QRS_NEXT_CUT()
PTP {E1 29336.998,E2 29336.998}
PTP {X 0,Y 607.858,A -85,B 0,C 180,E1 29336.998,E2 29336.998,E3 0,E4 0,E5 0,E6 0}
QRS_SPEED_INIT()
LIN {X 0,Y 607.858,Z 779,A -85,B 0,C 180,E1 29336.998,E2 29336.998,E3 0,E4 0,E5 0,E6 0} C_VEL
LIN {X 0,Y 607.858,Z 285.152,A -85,B 0,C 180,E1 29336.998,E2 29336.998} C_VEL
LIN {X 0,Y 607.858,Z 277.075,A -85,B 0,C 180,E1 29336.998,E2 29336.998} C_VEL
LIN {X 0,Y 607.845,Z 275.075,A -85,B 0,C 180,E1 29336.81,E2 29336.81} C_VEL
LIN {X 0,Y 607.872,Z 275.077,A -85,B 0,C 180,E1 29333.959,E2 29333.959} C_VEL
LIN {X 0,Y 607.849,Z 275.075,A -85,B 0,C 180,E1 29330.82,E2 29330.82} C_VEL
LIN {X 0,Y 607.873,Z 275.077,A -85,B 0,C 180,E1 29327.944,E2 29327.944} C_VEL
LIN {X 0,Y 607.848,Z 275.075,A -85,B 0,C 180,E1 29324.743,E2 29324.743} C_VEL
LIN {X 0,Y 607.877,Z 275.077,A -85,B 0,C 180,E1 29321.89,E2 29321.89} C_VEL
LIN {X 0,Y 607.853,Z 275.075,A -85,B 0,C 180,E1 29318.786,E2 29318.786} C_VEL
LIN {X 0,Y 607.875,Z 275.077,A -85,B 0,C 180,E1 29315.905,E2 29315.905} C_VEL
LIN {X 0,Y 607.85,Z 275.075,A -85,B 0,C 180,E1 29312.684,E2 29312.684} C_VEL
LIN {X 0,Y 607.895,Z 275.077,A -85,B 0,C 180,E1 29309.711,E2 29309.711} C_VEL
LIN {X 0,Y 607.853,Z 275.074,A -85,B 0,C 180,E1 29306.677,E2 29306.677} C_VEL
LIN {X 0,Y 607.897,Z 275.077,A -85,B 0,C 180,E1 29303.695,E2 29303.695} C_VEL
LIN {X 0,Y 607.852,Z 275.074,A -85,B 0,C 180,E1 29300.588,E2 29300.588} C_VEL
LIN {X 0,Y 607.905,Z 275.078,A -85,B 0,C 180,E1 29297.599,E2 29297.599} C_VEL
LIN {X 0,Y 607.851,Z 275.074,A -85,B 0,C 180,E1 29294.484,E2 29294.484} C_VEL
LIN {X 0,Y 607.918,Z 275.075,A -85,B 0,C 180,E1 29291.389,E2 29291.389} C_VEL
LIN {X 0,Y 607.852,Z 275.075,A -85,B 0,C 180,E1 29288.318,E2 29288.318} C_VEL
LIN {X 0,Y 607.91,Z 275.072,A -85,B 0,C 180,E1 29285.175,E2 29285.175} C_VEL
LIN {X 0,Y 607.858,Z 275.075,A -85,B 0,C 180,E1 29282.105,E2 29282.105} C_VEL
LIN {X 0,Y 607.887,Z 275.072,A -85,B 0,C 180,E1 29278.918,E2 29278.918} C_VEL
LIN {X 0,Y 607.867,Z 275.076,A -85,B 0,C 180,E1 29275.946,E2 29275.946} C_VEL
LIN {X 0,Y 607.866,Z 275.073,A -85,B 0,C 180,E1 29272.637,E2 29272.637} C_VEL
LIN {X 0,Y 607.899,Z 275.077,A -85,B 0,C 180,E1 29269.604,E2 29269.604} C_VEL
LIN {X 0,Y 607.859,Z 275.073,A -85,B 0,C 180,E1 29266.434,E2 29266.434} C_VEL
LIN {X 0,Y 607.914,Z 275.077,A -85,B 0,C 180,E1 29263.409,E2 29263.409} C_VEL
LIN {X 0,Y 607.859,Z 275.073,A -85,B 0,C 180,E1 29260.328,E2 29260.328} C_VEL
LIN {X 0,Y 607.917,Z 275.074,A -85,B 0,C 180,E1 29257.275,E2 29257.275} C_VEL
LIN {X 0,Y 607.859,Z 275.074,A -85,B 0,C 180,E1 29254.15,E2 29254.15} C_VEL
LIN {X 0,Y 607.912,Z 275.071,A -85,B 0,C 180,E1 29251.036,E2 29251.036} C_VEL
LIN {X 0,Y 607.868,Z 275.075,A -85,B 0,C 180,E1 29247.925,E2 29247.925} C_VEL
LIN {X 0,Y 607.888,Z 275.071,A -85,B 0,C 180,E1 29244.714,E2 29244.714} C_VEL
LIN {X 0,Y 607.885,Z 275.076,A -85,B 0,C 180,E1 29241.677,E2 29241.677} C_VEL
LIN {X 0,Y 607.869,Z 275.072,A -85,B 0,C 180,E1 29238.423,E2 29238.423} C_VEL
LIN {X 0,Y 607.918,Z 275.077,A -85,B 0,C 180,E1 29235.327,E2 29235.327} C_VEL
LIN {X 0,Y 607.865,Z 275.073,A -85,B 0,C 180,E1 29232.184,E2 29232.184} C_VEL
LIN {X 0,Y 607.915,Z 275.073,A -85,B 0,C 180,E1 29229.089,E2 29229.089} C_VEL
LIN {X 0,Y 607.866,Z 275.074,A -85,B 0,C 180,E1 29226.028,E2 29226.028} C_VEL
LIN {X 0,Y 607.913,Z 275.07,A -85,B 0,C 180,E1 29222.896,E2 29222.896} C_VEL
LIN {X 0,Y 607.876,Z 275.075,A -85,B 0,C 180,E1 29219.779,E2 29219.779} C_VEL
LIN {X 0,Y 607.884,Z 275.071,A -85,B 0,C 180,E1 29216.499,E2 29216.499} C_VEL
LIN {X 0,Y 607.915,Z 275.077,A -85,B 0,C 180,E1 29213.341,E2 29213.341} C_VEL
LIN {X 0,Y 607.871,Z 275.072,A -85,B 0,C 180,E1 29210.184,E2 29210.184} C_VEL
LIN {X 0,Y 607.913,Z 275.073,A -85,B 0,C 180,E1 29207.043,E2 29207.043} C_VEL
LIN {X 0,Y 607.872,Z 275.073,A -85,B 0,C 180,E1 29203.908,E2 29203.908} C_VEL
LIN {X 0,Y 607.915,Z 275.068,A -85,B 0,C 180,E1 29200.692,E2 29200.692} C_VEL
LIN {X 0,Y 607.896,Z 275.076,A -85,B 0,C 180,E1 29197.484,E2 29197.484} C_VEL
LIN {X 0,Y 607.878,Z 275.071,A -85,B 0,C 180,E1 29194.229,E2 29194.229} C_VEL
LIN {X 0,Y 607.914,Z 275.075,A -85,B 0,C 180,E1 29191.092,E2 29191.092} C_VEL
LIN {X 0,Y 607.874,Z 275.073,A -85,B 0,C 180,E1 29187.953,E2 29187.953} C_VEL
LIN {X 0,Y 607.888,Z 275.253,A -85,B 0,C 180,E1 29186.335,E2 29186.335} C_VEL
LIN {X 0,Y 607.91,Z 304.241,A -85,B 0,C 180,E1 29183.248,E2 29183.248} C_VEL
LIN {X 0,Y 607.905,Z 334.622,A -85,B 0,C 180,E1 29180.088,E2 29180.088} C_VEL
LIN {X 0,Y 607.882,Z 364.695,A -85,B 0,C 180,E1 29177.023,E2 29177.023} C_VEL
LIN {X 0,Y 607.92,Z 399.027,A -85,B 0,C 180,E1 29173.581,E2 29173.581} C_VEL
LIN {X 0,Y 607.897,Z 405.045,A -85,B 0,C 180,E1 29173.009,E2 29173.009} C_VEL
LIN {X 0,Y 607.911,Z 516.068,A -85,B 0,C 180,E1 29171.67,E2 29171.67} C_VEL
LIN {X 0,Y 607.905,Z 531.255,A -85,B 0,C 180,E1 29171.31,E2 29171.31} C_VEL
LIN {X 0,Y 607.911,Z 546.081,A -85,B 0,C 180,E1 29170.757,E2 29170.757} C_VEL
LIN {X 0,Y 607.897,Z 559.139,A -85,B 0,C 180,E1 29170.087,E2 29170.087} C_VEL
LIN {X 0,Y 607.919,Z 571.341,A -85,B 0,C 180,E1 29169.274,E2 29169.274} C_VEL
LIN {X 0,Y 607.919,Z 583.519,A -85,B 0,C 180,E1 29168.225,E2 29168.225} C_VEL
LIN {X 0,Y 607.919,Z 593.771,A -85,B 0,C 180,E1 29167.084,E2 29167.084} C_VEL
LIN {X 0,Y 607.917,Z 601.752,A -85,B 0,C 180,E1 29165.946,E2 29165.946} C_VEL
LIN {X 0,Y 607.914,Z 608.844,A -85,B 0,C 180,E1 29164.621,E2 29164.621} C_VEL
LIN {X 0,Y 607.917,Z 614.161,A -85,B 0,C 180,E1 29163.204,E2 29163.204} C_VEL
LIN {X 0,Y 607.915,Z 617.299,A -85,B 0,C 180,E1 29161.884,E2 29161.884} C_VEL
LIN {X 0,Y 607.918,Z 618.88,A -85,B 0,C 180,E1 29160.47,E2 29160.47} C_VEL
LIN {X 0,Y 607.915,Z 618.551,A -85,B 0,C 180,E1 29158.962,E2 29158.962} C_VEL
LIN {X 0,Y 607.916,Z 616.35,A -85,B 0,C 180,E1 29157.548,E2 29157.548} C_VEL
LIN {X 0,Y 607.918,Z 612.603,A -85,B 0,C 180,E1 29156.227,E2 29156.227} C_VEL
LIN {X 0,Y 607.917,Z 606.529,A -85,B 0,C 180,E1 29154.809,E2 29154.809} C_VEL
LIN {X 0,Y 607.918,Z 599.252,A -85,B 0,C 180,E1 29153.577,E2 29153.577} C_VEL
LIN {X 0,Y 607.918,Z 590.573,A -85,B 0,C 180,E1 29152.438,E2 29152.438} C_VEL
LIN {X 0,Y 607.919,Z 579.903,A -85,B 0,C 180,E1 29151.344,E2 29151.344} C_VEL
LIN {X 0,Y 607.911,Z 567.267,A -85,B 0,C 180,E1 29150.341,E2 29150.341} C_VEL
LIN {X 0,Y 607.909,Z 554.716,A -85,B 0,C 180,E1 29149.575,E2 29149.575} C_VEL
LIN {X 0,Y 607.907,Z 541.317,A -85,B 0,C 180,E1 29148.952,E2 29148.952} C_VEL
LIN {X 0,Y 607.913,Z 526.652,A -85,B 0,C 180,E1 29148.472,E2 29148.472} C_VEL
LIN {X 0,Y 607.902,Z 511.857,A -85,B 0,C 180,E1 29148.173,E2 29148.173} C_VEL
LIN {X 0,Y 607.896,Z 404.579,A -85,B 0,C 180,E1 29146.88,E2 29146.88} C_VEL
LIN {X 0,Y 607.909,Z 372.874,A -85,B 0,C 180,E1 29143.713,E2 29143.713} C_VEL
LIN {X 0,Y 607.9,Z 341.655,A -85,B 0,C 180,E1 29140.544,E2 29140.544} C_VEL
LIN {X 0,Y 607.843,Z 311.899,A -85,B 0,C 180,E1 29137.463,E2 29137.463} C_VEL
LIN {X 0,Y 607.918,Z 283.604,A -85,B 0,C 180,E1 29134.473,E2 29134.473} C_VEL
LIN {X 0,Y 607.859,Z 275.078,A -85,B 0,C 180,E1 29133.527,E2 29133.527} C_VEL
LIN {X 0,Y 607.916,Z 275.071,A -85,B 0,C 180,E1 29130.434,E2 29130.434} C_VEL
LIN {X 0,Y 607.895,Z 275.076,A -85,B 0,C 180,E1 29127.238,E2 29127.238} C_VEL
LIN {X 0,Y 607.897,Z 275.07,A -85,B 0,C 180,E1 29124.022,E2 29124.022} C_VEL
LIN {X 0,Y 607.901,Z 275.074,A -85,B 0,C 180,E1 29120.927,E2 29120.927} C_VEL
LIN {X 0,Y 607.902,Z 275.072,A -85,B 0,C 180,E1 29117.85,E2 29117.85} C_VEL
LIN {X 0,Y 607.886,Z 275.072,A -85,B 0,C 180,E1 29114.748,E2 29114.748} C_VEL
LIN {X 0,Y 607.905,Z 275.077,A -85,B 0,C 180,E1 29111.517,E2 29111.517} C_VEL
LIN {X 0,Y 607.903,Z 275.071,A -85,B 0,C 180,E1 29108.32,E2 29108.32} C_VEL
LIN {X 0,Y 607.854,Z 275.076,A -85,B 0,C 180,E1 29105.15,E2 29105.15} C_VEL
LIN {X 0,Y 607.918,Z 275.077,A -85,B 0,C 180,E1 29102.09,E2 29102.09} C_VEL
LIN {X 0,Y 607.866,Z 275.304,A -85,B 0,C 180,E1 29099.751,E2 29099.751} C_VEL
LIN {X 0,Y 607.899,Z 318.111,A -85,B 0,C 180,E1 29096.84,E2 29096.84} C_VEL
LIN {X 0,Y 607.901,Z 364.581,A -85,B 0,C 180,E1 29093.765,E2 29093.765} C_VEL
LIN {X 0,Y 607.908,Z 387.125,A -85,B 0,C 180,E1 29092.324,E2 29092.324} C_VEL
LIN {X 0,Y 607.914,Z 596.287,A -85,B 0,C 180,E1 29089.705,E2 29089.705} C_VEL
LIN {X 0,Y 607.913,Z 614.57,A -85,B 0,C 180,E1 29089.305,E2 29089.305} C_VEL
LIN {X 0,Y 607.915,Z 633.394,A -85,B 0,C 180,E1 29088.707,E2 29088.707} C_VEL
LIN {X 0,Y 607.916,Z 651.048,A -85,B 0,C 180,E1 29087.963,E2 29087.963} C_VEL
LIN {X 0,Y 607.919,Z 667.781,A -85,B 0,C 180,E1 29087.073,E2 29087.073} C_VEL
LIN {X 0,Y 607.916,Z 683.634,A -85,B 0,C 180,E1 29086.041,E2 29086.041} C_VEL
LIN {X 0,Y 607.917,Z 698.556,A -85,B 0,C 180,E1 29084.868,E2 29084.868} C_VEL
LIN {X 0,Y 607.918,Z 712.22,A -85,B 0,C 180,E1 29083.582,E2 29083.582} C_VEL
LIN {X 0,Y 607.916,Z 724.902,A -85,B 0,C 180,E1 29082.154,E2 29082.154} C_VEL
LIN {X 0,Y 607.911,Z 736.22,A -85,B 0,C 180,E1 29080.616,E2 29080.616} C_VEL
LIN {X 0,Y 607.92,Z 745.986,A -85,B 0,C 180,E1 29078.99,E2 29078.99} C_VEL
LIN {X 0,Y 607.913,Z 753.852,A -85,B 0,C 180,E1 29077.352,E2 29077.352} C_VEL
LIN {X 0,Y 607.906,Z 760.105,A -85,B 0,C 180,E1 29075.664,E2 29075.664} C_VEL
LIN {X 0,Y 607.917,Z 764.871,A -85,B 0,C 180,E1 29073.867,E2 29073.867} C_VEL
LIN {X 0,Y 607.911,Z 767.786,A -85,B 0,C 180,E1 29072.074,E2 29072.074} C_VEL
LIN {X 0,Y 607.907,Z 768.939,A -85,B 0,C 180,E1 29070.283,E2 29070.283} C_VEL
LIN {X 0,Y 607.916,Z 768.348,A -85,B 0,C 180,E1 29068.493,E2 29068.493} C_VEL
LIN {X 0,Y 607.908,Z 766.006,A -85,B 0,C 180,E1 29066.701,E2 29066.701} C_VEL
LIN {X 0,Y 607.918,Z 762.098,A -85,B 0,C 180,E1 29065,E2 29065} C_VEL
LIN {X 0,Y 607.91,Z 756.47,A -85,B 0,C 180,E1 29063.295,E2 29063.295} C_VEL
LIN {X 0,Y 607.914,Z 749.426,A -85,B 0,C 180,E1 29061.679,E2 29061.679} C_VEL
LIN {X 0,Y 607.914,Z 740.513,A -85,B 0,C 180,E1 29060.056,E2 29060.056} C_VEL
LIN {X 0,Y 607.919,Z 730.15,A -85,B 0,C 180,E1 29058.522,E2 29058.522} C_VEL
LIN {X 0,Y 607.915,Z 718.352,A -85,B 0,C 180,E1 29057.075,E2 29057.075} C_VEL
LIN {X 0,Y 607.915,Z 705.096,A -85,B 0,C 180,E1 29055.718,E2 29055.718} C_VEL
LIN {X 0,Y 607.917,Z 690.243,A -85,B 0,C 180,E1 29054.45,E2 29054.45} C_VEL
LIN {X 0,Y 607.917,Z 674.23,A -85,B 0,C 180,E1 29053.322,E2 29053.322} C_VEL
LIN {X 0,Y 607.911,Z 658.041,A -85,B 0,C 180,E1 29052.385,E2 29052.385} C_VEL
LIN {X 0,Y 607.913,Z 641.082,A -85,B 0,C 180,E1 29051.592,E2 29051.592} C_VEL
LIN {X 0,Y 607.916,Z 623.251,A -85,B 0,C 180,E1 29050.946,E2 29050.946} C_VEL
LIN {X 0,Y 607.91,Z 604.277,A -85,B 0,C 180,E1 29050.449,E2 29050.449} C_VEL
LIN {X 0,Y 607.914,Z 584.868,A -85,B 0,C 180,E1 29050.129,E2 29050.129} C_VEL
LIN {X 0,Y 607.907,Z 386.276,A -85,B 0,C 180,E1 29047.646,E2 29047.646} C_VEL
LIN {X 0,Y 607.897,Z 339.401,A -85,B 0,C 180,E1 29044.579,E2 29044.579} C_VEL
LIN {X 0,Y 607.883,Z 294.506,A -85,B 0,C 180,E1 29041.565,E2 29041.565} C_VEL
LIN {X 0,Y 607.864,Z 275.08,A -85,B 0,C 180,E1 29040.216,E2 29040.216} C_VEL
LIN {X 0,Y 607.84,Z 275.078,A -85,B 0,C 180,E1 29037.125,E2 29037.125} C_VEL
LIN {X 0,Y 607.847,Z 275.077,A -85,B 0,C 180,E1 29034.35,E2 29034.35} C_VEL
LIN {X 0,Y 607.837,Z 275.077,A -85,B 0,C 180,E1 29031.084,E2 29031.084} C_VEL
LIN {X 0,Y 607.854,Z 275.077,A -85,B 0,C 180,E1 29028.228,E2 29028.228} C_VEL
LIN {X 0,Y 607.833,Z 275.077,A -85,B 0,C 180,E1 29025.019,E2 29025.019} C_VEL
LIN {X 0,Y 607.849,Z 275.077,A -85,B 0,C 180,E1 29022.252,E2 29022.252} C_VEL
LIN {X 0,Y 607.838,Z 275.077,A -85,B 0,C 180,E1 29019.052,E2 29019.052} C_VEL
LIN {X 0,Y 607.843,Z 275.077,A -85,B 0,C 180,E1 29016.293,E2 29016.293} C_VEL
LIN {X 0,Y 607.845,Z 275.077,A -85,B 0,C 180,E1 29013.102,E2 29013.102} C_VEL
LIN {X 0,Y 607.842,Z 275.077,A -85,B 0,C 180,E1 29010.332,E2 29010.332} C_VEL
LIN {X 0,Y 607.84,Z 275.077,A -85,B 0,C 180,E1 29007.002,E2 29007.002} C_VEL
LIN {X 0,Y 607.846,Z 275.077,A -85,B 0,C 180,E1 29004.283,E2 29004.283} C_VEL
LIN {X 0,Y 607.845,Z 275.076,A -85,B 0,C 180,E1 29001.015,E2 29001.015} C_VEL
LIN {X 0,Y 607.851,Z 275.077,A -85,B 0,C 180,E1 28998.213,E2 28998.213} C_VEL
LIN {X 0,Y 607.845,Z 275.076,A -85,B 0,C 180,E1 28994.967,E2 28994.967} C_VEL
LIN {X 0,Y 607.847,Z 275.077,A -85,B 0,C 180,E1 28992.252,E2 28992.252} C_VEL
LIN {X 0,Y 607.85,Z 275.076,A -85,B 0,C 180,E1 28988.991,E2 28988.991} C_VEL
LIN {X 0,Y 607.849,Z 275.077,A -85,B 0,C 180,E1 28986.234,E2 28986.234} C_VEL
LIN {X 0,Y 607.849,Z 275.076,A -85,B 0,C 180,E1 28982.924,E2 28982.924} C_VEL
LIN {X 0,Y 607.859,Z 275.077,A -85,B 0,C 180,E1 28980.096,E2 28980.096} C_VEL
LIN {X 0,Y 607.85,Z 275.075,A -85,B 0,C 180,E1 28976.89,E2 28976.89} C_VEL
LIN {X 0,Y 607.845,Z 275.075,A -85,B 0,C 180,E1 28976.81,E2 28976.81} C_VEL
LIN {X 0,Y 606.844,Z 275.204,A -85,B 0,C 180,E1 28976.084,E2 28976.084} C_VEL
LIN {X 0,Y 600.488,Z 276.008,A -85,B 0,C 180,E1 28974.046,E2 28974.046} C_VEL
LIN {X 0,Y 599.975,Z 276.065,A -85,B 0,C 180,E1 28973.517,E2 28973.517} C_VEL
LIN {X 0,Y 599.903,Z 276.065,A -85,B 0,C 180,E1 28970.504,E2 28970.504} C_VEL
LIN {X 0,Y 599.969,Z 276.063,A -85,B 0,C 180,E1 28967.392,E2 28967.392} C_VEL
LIN {X 0,Y 599.907,Z 276.065,A -85,B 0,C 180,E1 28964.337,E2 28964.337} C_VEL
LIN {X 0,Y 599.95,Z 276.063,A -85,B 0,C 180,E1 28961.19,E2 28961.19} C_VEL
LIN {X 0,Y 599.909,Z 276.065,A -85,B 0,C 180,E1 28958.286,E2 28958.286} C_VEL
LIN {X 0,Y 599.952,Z 276.062,A -85,B 0,C 180,E1 28955.169,E2 28955.169} C_VEL
LIN {X 0,Y 599.914,Z 276.065,A -85,B 0,C 180,E1 28952.184,E2 28952.184} C_VEL
LIN {X 0,Y 599.928,Z 276.063,A -85,B 0,C 180,E1 28948.894,E2 28948.894} C_VEL
LIN {X 0,Y 599.932,Z 276.065,A -85,B 0,C 180,E1 28945.924,E2 28945.924} C_VEL
LIN {X 0,Y 599.921,Z 276.063,A -85,B 0,C 180,E1 28942.774,E2 28942.774} C_VEL
LIN {X 0,Y 599.94,Z 276.065,A -85,B 0,C 180,E1 28939.839,E2 28939.839} C_VEL
LIN {X 0,Y 599.915,Z 276.063,A -85,B 0,C 180,E1 28936.606,E2 28936.606} C_VEL
LIN {X 0,Y 599.972,Z 276.067,A -85,B 0,C 180,E1 28933.54,E2 28933.54} C_VEL
LIN {X 0,Y 599.913,Z 276.063,A -85,B 0,C 180,E1 28930.392,E2 28930.392} C_VEL
LIN {X 0,Y 599.977,Z 276.063,A -85,B 0,C 180,E1 28927.343,E2 28927.343} C_VEL
LIN {X 0,Y 599.915,Z 276.064,A -85,B 0,C 180,E1 28924.247,E2 28924.247} C_VEL
LIN {X 0,Y 599.968,Z 276.061,A -85,B 0,C 180,E1 28921.105,E2 28921.105} C_VEL
LIN {X 0,Y 599.923,Z 276.064,A -85,B 0,C 180,E1 28918.033,E2 28918.033} C_VEL
LIN {X 0,Y 599.933,Z 276.061,A -85,B 0,C 180,E1 28914.728,E2 28914.728} C_VEL
LIN {X 0,Y 599.948,Z 276.065,A -85,B 0,C 180,E1 28911.713,E2 28911.713} C_VEL
LIN {X 0,Y 599.923,Z 276.062,A -85,B 0,C 180,E1 28908.509,E2 28908.509} C_VEL
LIN {X 0,Y 599.975,Z 276.066,A -85,B 0,C 180,E1 28905.464,E2 28905.464} C_VEL
LIN {X 0,Y 599.92,Z 276.063,A -85,B 0,C 180,E1 28902.317,E2 28902.317} C_VEL
LIN {X 0,Y 599.978,Z 276.062,A -85,B 0,C 180,E1 28899.205,E2 28899.205} C_VEL
LIN {X 0,Y 599.922,Z 276.063,A -85,B 0,C 180,E1 28896.122,E2 28896.122} C_VEL
LIN {X 0,Y 599.971,Z 276.059,A -85,B 0,C 180,E1 28892.961,E2 28892.961} C_VEL
LIN {X 0,Y 599.93,Z 276.064,A -85,B 0,C 180,E1 28889.904,E2 28889.904} C_VEL
LIN {X 0,Y 599.939,Z 276.06,A -85,B 0,C 180,E1 28886.607,E2 28886.607} C_VEL
LIN {X 0,Y 599.965,Z 276.066,A -85,B 0,C 180,E1 28883.492,E2 28883.492} C_VEL
LIN {X 0,Y 599.926,Z 276.062,A -85,B 0,C 180,E1 28880.309,E2 28880.309} C_VEL
LIN {X 0,Y 599.977,Z 276.063,A -85,B 0,C 180,E1 28877.194,E2 28877.194} C_VEL
LIN {X 0,Y 599.926,Z 276.063,A -85,B 0,C 180,E1 28874.071,E2 28874.071} C_VEL
LIN {X 0,Y 599.974,Z 276.059,A -85,B 0,C 180,E1 28870.885,E2 28870.885} C_VEL
LIN {X 0,Y 599.938,Z 276.064,A -85,B 0,C 180,E1 28867.77,E2 28867.77} C_VEL
LIN {X 0,Y 599.937,Z 276.06,A -85,B 0,C 180,E1 28864.427,E2 28864.427} C_VEL
LIN {X 0,Y 599.974,Z 276.067,A -85,B 0,C 180,E1 28861.317,E2 28861.317} C_VEL
LIN {X 0,Y 599.929,Z 276.062,A -85,B 0,C 180,E1 28858.107,E2 28858.107} C_VEL
LIN {X 0,Y 599.975,Z 276.061,A -85,B 0,C 180,E1 28855.02,E2 28855.02} C_VEL
LIN {X 0,Y 599.933,Z 276.063,A -85,B 0,C 180,E1 28851.869,E2 28851.869} C_VEL
LIN {X 0,Y 599.968,Z 276.058,A -85,B 0,C 180,E1 28848.704,E2 28848.704} C_VEL
LIN {X 0,Y 599.957,Z 276.065,A -85,B 0,C 180,E1 28845.499,E2 28845.499} C_VEL
LIN {X 0,Y 599.938,Z 276.06,A -85,B 0,C 180,E1 28842.27,E2 28842.27} C_VEL
LIN {X 0,Y 599.977,Z 276.065,A -85,B 0,C 180,E1 28839.166,E2 28839.166} C_VEL
LIN {X 0,Y 599.934,Z 276.062,A -85,B 0,C 180,E1 28836.035,E2 28836.035} C_VEL
LIN {X 0,Y 599.974,Z 276.06,A -85,B 0,C 180,E1 28832.868,E2 28832.868} C_VEL
LIN {X 0,Y 599.94,Z 276.064,A -85,B 0,C 180,E1 28829.738,E2 28829.738} C_VEL
LIN {X 0,Y 599.997,Z 276.241,A -85,B 0,C 180,E1 28826.601,E2 28826.601} C_VEL
LIN {X 0,Y 600.264,Z 284.48,A -85,B 0,C 180,E1 28825.69,E2 28825.69} C_VEL
LIN {X 0,Y 600.192,Z 314.246,A -85,B 0,C 180,E1 28822.501,E2 28822.501} C_VEL
LIN {X 0,Y 600.105,Z 344.224,A -85,B 0,C 180,E1 28819.362,E2 28819.362} C_VEL
LIN {X 0,Y 600.059,Z 375.427,A -85,B 0,C 180,E1 28816.155,E2 28816.155} C_VEL
LIN {X 0,Y 600.035,Z 405.097,A -85,B 0,C 180,E1 28813.182,E2 28813.182} C_VEL
LIN {X 0,Y 600.074,Z 516.391,A -85,B 0,C 180,E1 28811.819,E2 28811.819} C_VEL
LIN {X 0,Y 600.051,Z 531.275,A -85,B 0,C 180,E1 28811.46,E2 28811.46} C_VEL
LIN {X 0,Y 600.03,Z 546.096,A -85,B 0,C 180,E1 28810.9,E2 28810.9} C_VEL
LIN {X 0,Y 599.988,Z 559.151,A -85,B 0,C 180,E1 28810.221,E2 28810.221} C_VEL
LIN {X 0,Y 599.986,Z 571.349,A -85,B 0,C 180,E1 28809.398,E2 28809.398} C_VEL
LIN {X 0,Y 599.961,Z 583.526,A -85,B 0,C 180,E1 28808.335,E2 28808.335} C_VEL
LIN {X 0,Y 599.942,Z 593.776,A -85,B 0,C 180,E1 28807.179,E2 28807.179} C_VEL
LIN {X 0,Y 599.928,Z 601.756,A -85,B 0,C 180,E1 28806.026,E2 28806.026} C_VEL
LIN {X 0,Y 599.919,Z 608.863,A -85,B 0,C 180,E1 28804.679,E2 28804.679} C_VEL
LIN {X 0,Y 599.92,Z 614.164,A -85,B 0,C 180,E1 28803.247,E2 28803.247} C_VEL
LIN {X 0,Y 599.916,Z 617.301,A -85,B 0,C 180,E1 28801.909,E2 28801.909} C_VEL
LIN {X 0,Y 599.919,Z 618.88,A -85,B 0,C 180,E1 28800.476,E2 28800.476} C_VEL
LIN {X 0,Y 599.915,Z 618.55,A -85,B 0,C 180,E1 28798.948,E2 28798.948} C_VEL
LIN {X 0,Y 599.917,Z 616.349,A -85,B 0,C 180,E1 28797.515,E2 28797.515} C_VEL
LIN {X 0,Y 599.919,Z 612.601,A -85,B 0,C 180,E1 28796.176,E2 28796.176} C_VEL
LIN {X 0,Y 599.923,Z 606.526,A -85,B 0,C 180,E1 28794.739,E2 28794.739} C_VEL
LIN {X 0,Y 599.933,Z 599.249,A -85,B 0,C 180,E1 28793.491,E2 28793.491} C_VEL
LIN {X 0,Y 599.948,Z 590.568,A -85,B 0,C 180,E1 28792.337,E2 28792.337} C_VEL
LIN {X 0,Y 599.97,Z 579.677,A -85,B 0,C 180,E1 28791.208,E2 28791.208} C_VEL
LIN {X 0,Y 599.983,Z 567.257,A -85,B 0,C 180,E1 28790.212,E2 28790.212} C_VEL
LIN {X 0,Y 600.012,Z 554.707,A -85,B 0,C 180,E1 28789.437,E2 28789.437} C_VEL
LIN {X 0,Y 600.037,Z 541.302,A -85,B 0,C 180,E1 28788.805,E2 28788.805} C_VEL
LIN {X 0,Y 600.064,Z 525.867,A -85,B 0,C 180,E1 28788.297,E2 28788.297} C_VEL
LIN {X 0,Y 600.069,Z 510.599,A -85,B 0,C 180,E1 28787.999,E2 28787.999} C_VEL
LIN {X 0,Y 600.001,Z 404.573,A -85,B 0,C 180,E1 28786.704,E2 28786.704} C_VEL
LIN {X 0,Y 600.055,Z 372.38,A -85,B 0,C 180,E1 28783.444,E2 28783.444} C_VEL
LIN {X 0,Y 600.14,Z 341.577,A -85,B 0,C 180,E1 28780.275,E2 28780.275} C_VEL
LIN {X 0,Y 600.139,Z 312.38,A -85,B 0,C 180,E1 28777.209,E2 28777.209} C_VEL
LIN {X 0,Y 600.29,Z 284.085,A -85,B 0,C 180,E1 28774.178,E2 28774.178} C_VEL
LIN {X 0,Y 600.043,Z 276.767,A -85,B 0,C 180,E1 28773.368,E2 28773.368} C_VEL
LIN {X 0,Y 599.929,Z 276.07,A -85,B 0,C 180,E1 28773.256,E2 28773.256} C_VEL
LIN {X 0,Y 599.947,Z 276.061,A -85,B 0,C 180,E1 28770.001,E2 28770.001} C_VEL
LIN {X 0,Y 599.974,Z 276.065,A -85,B 0,C 180,E1 28766.864,E2 28766.864} C_VEL
LIN {X 0,Y 599.951,Z 276.062,A -85,B 0,C 180,E1 28763.726,E2 28763.726} C_VEL
LIN {X 0,Y 599.962,Z 276.06,A -85,B 0,C 180,E1 28760.583,E2 28760.583} C_VEL
LIN {X 0,Y 599.968,Z 276.066,A -85,B 0,C 180,E1 28757.302,E2 28757.302} C_VEL
LIN {X 0,Y 599.974,Z 276.059,A -85,B 0,C 180,E1 28754.088,E2 28754.088} C_VEL
LIN {X 0,Y 599.935,Z 276.063,A -85,B 0,C 180,E1 28750.919,E2 28750.919} C_VEL
LIN {X 0,Y 599.968,Z 276.067,A -85,B 0,C 180,E1 28747.707,E2 28747.707} C_VEL
LIN {X 0,Y 599.93,Z 276.064,A -85,B 0,C 180,E1 28744.634,E2 28744.634} C_VEL
LIN {X 0,Y 599.909,Z 276.068,A -85,B 0,C 180,E1 28741.422,E2 28741.422} C_VEL
LIN {X 0,Y 599.972,Z 276.106,A -85,B 0,C 180,E1 28740.126,E2 28740.126} C_VEL
LIN {X 0,Y 600.585,Z 279.631,A -85,B 0,C 180,E1 28739.846,E2 28739.846} C_VEL
LIN {X 0,Y 600.503,Z 321.261,A -85,B 0,C 180,E1 28736.983,E2 28736.983} C_VEL
LIN {X 0,Y 600.374,Z 367.732,A -85,B 0,C 180,E1 28733.872,E2 28733.872} C_VEL
LIN {X 0,Y 600.412,Z 387.17,A -85,B 0,C 180,E1 28732.618,E2 28732.618} C_VEL
LIN {X 0,Y 600.374,Z 596.287,A -85,B 0,C 180,E1 28729.963,E2 28729.963} C_VEL
LIN {X 0,Y 600.333,Z 615.274,A -85,B 0,C 180,E1 28729.539,E2 28729.539} C_VEL
LIN {X 0,Y 600.287,Z 633.392,A -85,B 0,C 180,E1 28728.954,E2 28728.954} C_VEL
LIN {X 0,Y 600.233,Z 651.044,A -85,B 0,C 180,E1 28728.201,E2 28728.201} C_VEL
LIN {X 0,Y 600.179,Z 667.696,A -85,B 0,C 180,E1 28727.305,E2 28727.305} C_VEL
LIN {X 0,Y 600.122,Z 683.632,A -85,B 0,C 180,E1 28726.255,E2 28726.255} C_VEL
LIN {X 0,Y 600.069,Z 698.557,A -85,B 0,C 180,E1 28725.067,E2 28725.067} C_VEL
LIN {X 0,Y 600.02,Z 712.014,A -85,B 0,C 180,E1 28723.786,E2 28723.786} C_VEL
LIN {X 0,Y 599.982,Z 724.903,A -85,B 0,C 180,E1 28722.317,E2 28722.317} C_VEL
LIN {X 0,Y 599.953,Z 736.221,A -85,B 0,C 180,E1 28720.758,E2 28720.758} C_VEL
LIN {X 0,Y 599.939,Z 745.987,A -85,B 0,C 180,E1 28719.111,E2 28719.111} C_VEL
LIN {X 0,Y 599.923,Z 754.034,A -85,B 0,C 180,E1 28717.407,E2 28717.407} C_VEL
LIN {X 0,Y 599.91,Z 760.408,A -85,B 0,C 180,E1 28715.644,E2 28715.644} C_VEL
LIN {X 0,Y 599.918,Z 764.872,A -85,B 0,C 180,E1 28713.919,E2 28713.919} C_VEL
LIN {X 0,Y 599.911,Z 767.787,A -85,B 0,C 180,E1 28712.102,E2 28712.102} C_VEL
LIN {X 0,Y 599.907,Z 768.939,A -85,B 0,C 180,E1 28710.287,E2 28710.287} C_VEL
LIN {X 0,Y 599.915,Z 768.349,A -85,B 0,C 180,E1 28708.473,E2 28708.473} C_VEL
LIN {X 0,Y 599.907,Z 766.006,A -85,B 0,C 180,E1 28706.657,E2 28706.657} C_VEL
LIN {X 0,Y 599.92,Z 762.098,A -85,B 0,C 180,E1 28704.933,E2 28704.933} C_VEL
LIN {X 0,Y 599.919,Z 756.47,A -85,B 0,C 180,E1 28703.205,E2 28703.205} C_VEL
LIN {X 0,Y 599.927,Z 749.427,A -85,B 0,C 180,E1 28701.567,E2 28701.567} C_VEL
LIN {X 0,Y 599.947,Z 740.515,A -85,B 0,C 180,E1 28699.923,E2 28699.923} C_VEL
LIN {X 0,Y 599.969,Z 730.151,A -85,B 0,C 180,E1 28698.367,E2 28698.367} C_VEL
LIN {X 0,Y 600.001,Z 718.353,A -85,B 0,C 180,E1 28696.902,E2 28696.902} C_VEL
LIN {X 0,Y 600.046,Z 704.766,A -85,B 0,C 180,E1 28695.494,E2 28695.494} C_VEL
LIN {X 0,Y 600.103,Z 690.243,A -85,B 0,C 180,E1 28694.242,E2 28694.242} C_VEL
LIN {X 0,Y 600.165,Z 674.233,A -85,B 0,C 180,E1 28693.1,E2 28693.1} C_VEL
LIN {X 0,Y 600.216,Z 657.049,A -85,B 0,C 180,E1 28692.102,E2 28692.102} C_VEL
LIN {X 0,Y 600.277,Z 639.677,A -85,B 0,C 180,E1 28691.294,E2 28691.294} C_VEL
LIN {X 0,Y 600.33,Z 621.682,A -85,B 0,C 180,E1 28690.649,E2 28690.649} C_VEL
LIN {X 0,Y 600.361,Z 603.347,A -85,B 0,C 180,E1 28690.174,E2 28690.174} C_VEL
LIN {X 0,Y 600.389,Z 583.667,A -85,B 0,C 180,E1 28689.854,E2 28689.854} C_VEL
LIN {X 0,Y 600.335,Z 386.634,A -85,B 0,C 180,E1 28687.372,E2 28687.372} C_VEL
LIN {X 0,Y 600.446,Z 340.976,A -85,B 0,C 180,E1 28684.346,E2 28684.346} C_VEL
LIN {X 0,Y 600.565,Z 296.568,A -85,B 0,C 180,E1 28681.329,E2 28681.329} C_VEL
LIN {X 0,Y 600.426,Z 277.965,A -85,B 0,C 180,E1 28680.029,E2 28680.029} C_VEL
LIN {X 0,Y 599.967,Z 276.066,A -85,B 0,C 180,E1 28679.844,E2 28679.844} C_VEL
LIN {X 0,Y 599.891,Z 276.067,A -85,B 0,C 180,E1 28676.794,E2 28676.794} C_VEL
LIN {X 0,Y 599.96,Z 276.068,A -85,B 0,C 180,E1 28673.729,E2 28673.729} C_VEL
LIN {X 0,Y 599.89,Z 276.067,A -85,B 0,C 180,E1 28670.809,E2 28670.809} C_VEL
LIN {X 0,Y 599.966,Z 276.067,A -85,B 0,C 180,E1 28667.681,E2 28667.681} C_VEL
LIN {X 0,Y 599.889,Z 276.067,A -85,B 0,C 180,E1 28664.698,E2 28664.698} C_VEL
LIN {X 0,Y 599.969,Z 276.067,A -85,B 0,C 180,E1 28661.678,E2 28661.678} C_VEL
LIN {X 0,Y 599.89,Z 276.066,A -85,B 0,C 180,E1 28658.685,E2 28658.685} C_VEL
LIN {X 0,Y 599.975,Z 276.066,A -85,B 0,C 180,E1 28655.682,E2 28655.682} C_VEL
LIN {X 0,Y 599.893,Z 276.066,A -85,B 0,C 180,E1 28652.572,E2 28652.572} C_VEL
LIN {X 0,Y 599.946,Z 276.065,A -85,B 0,C 180,E1 28649.449,E2 28649.449} C_VEL
LIN {X 0,Y 599.896,Z 276.066,A -85,B 0,C 180,E1 28646.49,E2 28646.49} C_VEL
LIN {X 0,Y 599.94,Z 276.065,A -85,B 0,C 180,E1 28643.37,E2 28643.37} C_VEL
LIN {X 0,Y 599.901,Z 276.066,A -85,B 0,C 180,E1 28640.387,E2 28640.387} C_VEL
LIN {X 0,Y 599.92,Z 276.065,A -85,B 0,C 180,E1 28637.158,E2 28637.158} C_VEL
LIN {X 0,Y 599.907,Z 276.066,A -85,B 0,C 180,E1 28634.282,E2 28634.282} C_VEL
LIN {X 0,Y 599.908,Z 276.065,A -85,B 0,C 180,E1 28630.954,E2 28630.954} C_VEL
LIN {X 0,Y 599.919,Z 276.066,A -85,B 0,C 180,E1 28628.12,E2 28628.12} C_VEL
LIN {X 0,Y 599.906,Z 276.065,A -85,B 0,C 180,E1 28624.877,E2 28624.877} C_VEL
LIN {X 0,Y 599.929,Z 276.066,A -85,B 0,C 180,E1 28622.007,E2 28622.007} C_VEL
LIN {X 0,Y 599.908,Z 276.064,A -85,B 0,C 180,E1 28618.855,E2 28618.855} C_VEL
LIN {X 0,Y 599.93,Z 276.066,A -85,B 0,C 180,E1 28615.988,E2 28615.988} C_VEL
LIN {X 0,Y 599.975,Z 276.065,A -85,B 0,C 180,E1 28613.517,E2 28613.517} C_VEL
LIN {X 0,Y 598.985,Z 276.182,A -85,B 0,C 180,E1 28612.781,E2 28612.781} C_VEL
LIN {X 0,Y 592.49,Z 276.989,A -85,B 0,C 180,E1 28610.718,E2 28610.718} C_VEL
LIN {X 0,Y 591.975,Z 277.054,A -85,B 0,C 180,E1 28610.18,E2 28610.18} C_VEL
LIN {X 0,Y 591.974,Z 277.053,A -85,B 0,C 180,E1 28606.821,E2 28606.821} C_VEL
LIN {X 0,Y 591.996,Z 277.055,A -85,B 0,C 180,E1 28603.921,E2 28603.921} C_VEL
LIN {X 0,Y 591.97,Z 277.053,A -85,B 0,C 180,E1 28600.669,E2 28600.669} C_VEL
LIN {X 0,Y 592.039,Z 277.055,A -85,B 0,C 180,E1 28597.564,E2 28597.564} C_VEL
LIN {X 0,Y 591.968,Z 277.053,A -85,B 0,C 180,E1 28594.413,E2 28594.413} C_VEL
LIN {X 0,Y 592.034,Z 277.052,A -85,B 0,C 180,E1 28591.341,E2 28591.341} C_VEL
LIN {X 0,Y 591.971,Z 277.053,A -85,B 0,C 180,E1 28588.315,E2 28588.315} C_VEL
LIN {X 0,Y 592.019,Z 277.051,A -85,B 0,C 180,E1 28585.164,E2 28585.164} C_VEL
LIN {X 0,Y 591.976,Z 277.053,A -85,B 0,C 180,E1 28582.188,E2 28582.188} C_VEL
LIN {X 0,Y 591.998,Z 277.051,A -85,B 0,C 180,E1 28578.931,E2 28578.931} C_VEL
LIN {X 0,Y 591.984,Z 277.054,A -85,B 0,C 180,E1 28576.013,E2 28576.013} C_VEL
LIN {X 0,Y 591.984,Z 277.051,A -85,B 0,C 180,E1 28572.72,E2 28572.72} C_VEL
LIN {X 0,Y 592.023,Z 277.055,A -85,B 0,C 180,E1 28569.638,E2 28569.638} C_VEL
LIN {X 0,Y 591.976,Z 277.052,A -85,B 0,C 180,E1 28566.478,E2 28566.478} C_VEL
LIN {X 0,Y 592.038,Z 277.054,A -85,B 0,C 180,E1 28563.404,E2 28563.404} C_VEL
LIN {X 0,Y 591.976,Z 277.052,A -85,B 0,C 180,E1 28560.331,E2 28560.331} C_VEL
LIN {X 0,Y 592.04,Z 277.05,A -85,B 0,C 180,E1 28557.236,E2 28557.236} C_VEL
LIN {X 0,Y 591.981,Z 277.053,A -85,B 0,C 180,E1 28554.125,E2 28554.125} C_VEL
LIN {X 0,Y 592.018,Z 277.049,A -85,B 0,C 180,E1 28550.946,E2 28550.946} C_VEL
LIN {X 0,Y 591.992,Z 277.053,A -85,B 0,C 180,E1 28547.901,E2 28547.901} C_VEL
LIN {X 0,Y 591.989,Z 277.051,A -85,B 0,C 180,E1 28544.575,E2 28544.575} C_VEL
LIN {X 0,Y 592.032,Z 277.055,A -85,B 0,C 180,E1 28541.494,E2 28541.494} C_VEL
LIN {X 0,Y 591.982,Z 277.051,A -85,B 0,C 180,E1 28538.351,E2 28538.351} C_VEL
LIN {X 0,Y 592.039,Z 277.052,A -85,B 0,C 180,E1 28535.232,E2 28535.232} C_VEL
LIN {X 0,Y 591.984,Z 277.052,A -85,B 0,C 180,E1 28532.129,E2 28532.129} C_VEL
LIN {X 0,Y 592.029,Z 277.049,A -85,B 0,C 180,E1 28528.935,E2 28528.935} C_VEL
LIN {X 0,Y 591.996,Z 277.053,A -85,B 0,C 180,E1 28525.834,E2 28525.834} C_VEL
LIN {X 0,Y 591.993,Z 277.05,A -85,B 0,C 180,E1 28522.471,E2 28522.471} C_VEL
LIN {X 0,Y 592.036,Z 277.056,A -85,B 0,C 180,E1 28519.377,E2 28519.377} C_VEL
LIN {X 0,Y 591.986,Z 277.051,A -85,B 0,C 180,E1 28516.197,E2 28516.197} C_VEL
LIN {X 0,Y 592.038,Z 277.051,A -85,B 0,C 180,E1 28513.113,E2 28513.113} C_VEL
LIN {X 0,Y 591.991,Z 277.052,A -85,B 0,C 180,E1 28509.948,E2 28509.948} C_VEL
LIN {X 0,Y 592.023,Z 277.048,A -85,B 0,C 180,E1 28506.721,E2 28506.721} C_VEL
LIN {X 0,Y 592.02,Z 277.054,A -85,B 0,C 180,E1 28503.517,E2 28503.517} C_VEL
LIN {X 0,Y 591.996,Z 277.049,A -85,B 0,C 180,E1 28500.338,E2 28500.338} C_VEL
LIN {X 0,Y 592.038,Z 277.052,A -85,B 0,C 180,E1 28497.171,E2 28497.171} C_VEL
LIN {X 0,Y 591.992,Z 277.051,A -85,B 0,C 180,E1 28493.996,E2 28493.996} C_VEL
LIN {X 0,Y 592.038,Z 277.047,A -85,B 0,C 180,E1 28490.817,E2 28490.817} C_VEL
LIN {X 0,Y 592.007,Z 277.053,A -85,B 0,C 180,E1 28487.632,E2 28487.632} C_VEL
LIN {X 0,Y 592.005,Z 277.048,A -85,B 0,C 180,E1 28484.361,E2 28484.361} C_VEL
LIN {X 0,Y 592.037,Z 277.054,A -85,B 0,C 180,E1 28481.194,E2 28481.194} C_VEL
LIN {X 0,Y 591.995,Z 277.051,A -85,B 0,C 180,E1 28478.056,E2 28478.056} C_VEL
LIN {X 0,Y 592.036,Z 277.05,A -85,B 0,C 180,E1 28474.923,E2 28474.923} C_VEL
LIN {X 0,Y 591.997,Z 277.052,A -85,B 0,C 180,E1 28471.798,E2 28471.798} C_VEL
LIN {X 0,Y 592.029,Z 277.049,A -85,B 0,C 180,E1 28468.549,E2 28468.549} C_VEL
LIN {X 0,Y 592.046,Z 277.139,A -85,B 0,C 180,E1 28466.89,E2 28466.89} C_VEL
LIN {X 0,Y 592.666,Z 281.437,A -85,B 0,C 180,E1 28466.384,E2 28466.384} C_VEL
LIN {X 0,Y 592.523,Z 309.616,A -85,B 0,C 180,E1 28463.308,E2 28463.308} C_VEL
LIN {X 0,Y 592.379,Z 340.33,A -85,B 0,C 180,E1 28460.036,E2 28460.036} C_VEL
LIN {X 0,Y 592.241,Z 372.02,A -85,B 0,C 180,E1 28456.727,E2 28456.727} C_VEL
LIN {X 0,Y 592.11,Z 404.162,A -85,B 0,C 180,E1 28453.428,E2 28453.428} C_VEL
LIN {X 0,Y 592.176,Z 405.374,A -85,B 0,C 180,E1 28453.358,E2 28453.358} C_VEL
LIN {X 0,Y 592.241,Z 516.485,A -85,B 0,C 180,E1 28451.977,E2 28451.977} C_VEL
LIN {X 0,Y 592.201,Z 531.295,A -85,B 0,C 180,E1 28451.614,E2 28451.614} C_VEL
LIN {X 0,Y 592.153,Z 546.112,A -85,B 0,C 180,E1 28451.047,E2 28451.047} C_VEL
LIN {X 0,Y 592.084,Z 559.163,A -85,B 0,C 180,E1 28450.359,E2 28450.359} C_VEL
LIN {X 0,Y 592.057,Z 571.56,A -85,B 0,C 180,E1 28449.509,E2 28449.509} C_VEL
LIN {X 0,Y 592.006,Z 583.532,A -85,B 0,C 180,E1 28448.448,E2 28448.448} C_VEL
LIN {X 0,Y 591.966,Z 593.78,A -85,B 0,C 180,E1 28447.276,E2 28447.276} C_VEL
LIN {X 0,Y 591.94,Z 601.761,A -85,B 0,C 180,E1 28446.107,E2 28446.107} C_VEL
LIN {X 0,Y 591.926,Z 608.849,A -85,B 0,C 180,E1 28444.746,E2 28444.746} C_VEL
LIN {X 0,Y 591.922,Z 614.166,A -85,B 0,C 180,E1 28443.291,E2 28443.291} C_VEL
LIN {X 0,Y 591.916,Z 617.302,A -85,B 0,C 180,E1 28441.935,E2 28441.935} C_VEL
LIN {X 0,Y 591.919,Z 618.881,A -85,B 0,C 180,E1 28440.483,E2 28440.483} C_VEL
LIN {X 0,Y 591.914,Z 618.549,A -85,B 0,C 180,E1 28438.934,E2 28438.934} C_VEL
LIN {X 0,Y 591.918,Z 616.348,A -85,B 0,C 180,E1 28437.482,E2 28437.482} C_VEL
LIN {X 0,Y 591.921,Z 612.599,A -85,B 0,C 180,E1 28436.124,E2 28436.124} C_VEL
LIN {X 0,Y 591.93,Z 606.523,A -85,B 0,C 180,E1 28434.668,E2 28434.668} C_VEL
LIN {X 0,Y 591.948,Z 599.245,A -85,B 0,C 180,E1 28433.403,E2 28433.403} C_VEL
LIN {X 0,Y 591.978,Z 590.562,A -85,B 0,C 180,E1 28432.233,E2 28432.233} C_VEL
LIN {X 0,Y 592.021,Z 579.978,A -85,B 0,C 180,E1 28431.118,E2 28431.118} C_VEL
LIN {X 0,Y 592.059,Z 567.611,A -85,B 0,C 180,E1 28430.107,E2 28430.107} C_VEL
LIN {X 0,Y 592.118,Z 554.698,A -85,B 0,C 180,E1 28429.294,E2 28429.294} C_VEL
LIN {X 0,Y 592.169,Z 541.288,A -85,B 0,C 180,E1 28428.654,E2 28428.654} C_VEL
LIN {X 0,Y 592.222,Z 525.844,A -85,B 0,C 180,E1 28428.14,E2 28428.14} C_VEL
LIN {X 0,Y 592.241,Z 510.445,A -85,B 0,C 180,E1 28427.837,E2 28427.837} C_VEL
LIN {X 0,Y 592.11,Z 404.676,A -85,B 0,C 180,E1 28426.534,E2 28426.534} C_VEL
LIN {X 0,Y 592.212,Z 372.16,A -85,B 0,C 180,E1 28423.196,E2 28423.196} C_VEL
LIN {X 0,Y 592.373,Z 341.643,A -85,B 0,C 180,E1 28420.013,E2 28420.013} C_VEL
LIN {X 0,Y 592.446,Z 312.861,A -85,B 0,C 180,E1 28416.949,E2 28416.949} C_VEL
LIN {X 0,Y 592.666,Z 283.64,A -85,B 0,C 180,E1 28413.767,E2 28413.767} C_VEL
LIN {X 0,Y 592.44,Z 278.875,A -85,B 0,C 180,E1 28413.216,E2 28413.216} C_VEL
LIN {X 0,Y 592.013,Z 277.059,A -85,B 0,C 180,E1 28412.978,E2 28412.978} C_VEL
LIN {X 0,Y 591.999,Z 277.052,A -85,B 0,C 180,E1 28409.78,E2 28409.78} C_VEL
LIN {X 0,Y 592.033,Z 277.052,A -85,B 0,C 180,E1 28406.709,E2 28406.709} C_VEL
LIN {X 0,Y 592.018,Z 277.053,A -85,B 0,C 180,E1 28403.507,E2 28403.507} C_VEL
LIN {X 0,Y 592.036,Z 277.046,A -85,B 0,C 180,E1 28400.202,E2 28400.202} C_VEL
LIN {X 0,Y 592.014,Z 277.052,A -85,B 0,C 180,E1 28396.974,E2 28396.974} C_VEL
LIN {X 0,Y 592.033,Z 277.052,A -85,B 0,C 180,E1 28393.824,E2 28393.824} C_VEL
LIN {X 0,Y 592.002,Z 277.051,A -85,B 0,C 180,E1 28390.682,E2 28390.682} C_VEL
LIN {X 0,Y 591.993,Z 277.055,A -85,B 0,C 180,E1 28387.326,E2 28387.326} C_VEL
LIN {X 0,Y 592.039,Z 277.054,A -85,B 0,C 180,E1 28384.153,E2 28384.153} C_VEL
LIN {X 0,Y 591.962,Z 277.058,A -85,B 0,C 180,E1 28381.09,E2 28381.09} C_VEL
LIN {X 0,Y 591.995,Z 277.069,A -85,B 0,C 180,E1 28380.506,E2 28380.506} C_VEL
LIN {X 0,Y 593.329,Z 281.88,A -85,B 0,C 180,E1 28380.089,E2 28380.089} C_VEL
LIN {X 0,Y 593.114,Z 323.624,A -85,B 0,C 180,E1 28377.184,E2 28377.184} C_VEL
LIN {X 0,Y 592.86,Z 369.307,A -85,B 0,C 180,E1 28374.088,E2 28374.088} C_VEL
LIN {X 0,Y 592.853,Z 387.15,A -85,B 0,C 180,E1 28372.923,E2 28372.923} C_VEL
LIN {X 0,Y 593.11,Z 400.207,A -85,B 0,C 180,E1 28372.744,E2 28372.744} C_VEL
LIN {X 0,Y 592.848,Z 596.287,A -85,B 0,C 180,E1 28370.228,E2 28370.228} C_VEL
LIN {X 0,Y 592.769,Z 615.285,A -85,B 0,C 180,E1 28369.798,E2 28369.798} C_VEL
LIN {X 0,Y 592.678,Z 633.389,A -85,B 0,C 180,E1 28369.207,E2 28369.207} C_VEL
LIN {X 0,Y 592.57,Z 651.041,A -85,B 0,C 180,E1 28368.444,E2 28368.444} C_VEL
LIN {X 0,Y 592.459,Z 667.7,A -85,B 0,C 180,E1 28367.538,E2 28367.538} C_VEL
LIN {X 0,Y 592.342,Z 683.629,A -85,B 0,C 180,E1 28366.475,E2 28366.475} C_VEL
LIN {X 0,Y 592.23,Z 698.556,A -85,B 0,C 180,E1 28365.271,E2 28365.271} C_VEL
LIN {X 0,Y 592.131,Z 712.013,A -85,B 0,C 180,E1 28363.974,E2 28363.974} C_VEL
LIN {X 0,Y 592.057,Z 724.421,A -85,B 0,C 180,E1 28362.546,E2 28362.546} C_VEL
LIN {X 0,Y 592.002,Z 735.584,A -85,B 0,C 180,E1 28361.003,E2 28361.003} C_VEL
LIN {X 0,Y 591.956,Z 745.471,A -85,B 0,C 180,E1 28359.332,E2 28359.332} C_VEL
LIN {X 0,Y 591.936,Z 753.77,A -85,B 0,C 180,E1 28357.572,E2 28357.572} C_VEL
LIN {X 0,Y 591.913,Z 760.265,A -85,B 0,C 180,E1 28355.767,E2 28355.767} C_VEL
LIN {X 0,Y 591.918,Z 764.872,A -85,B 0,C 180,E1 28353.972,E2 28353.972} C_VEL
LIN {X 0,Y 591.911,Z 767.788,A -85,B 0,C 180,E1 28352.13,E2 28352.13} C_VEL
LIN {X 0,Y 591.908,Z 768.939,A -85,B 0,C 180,E1 28350.291,E2 28350.291} C_VEL
LIN {X 0,Y 591.914,Z 768.349,A -85,B 0,C 180,E1 28348.452,E2 28348.452} C_VEL
LIN {X 0,Y 591.907,Z 766.007,A -85,B 0,C 180,E1 28346.611,E2 28346.611} C_VEL
LIN {X 0,Y 591.921,Z 762.099,A -85,B 0,C 180,E1 28344.864,E2 28344.864} C_VEL
LIN {X 0,Y 591.93,Z 756.47,A -85,B 0,C 180,E1 28343.113,E2 28343.113} C_VEL
LIN {X 0,Y 591.94,Z 749.428,A -85,B 0,C 180,E1 28341.453,E2 28341.453} C_VEL
LIN {X 0,Y 591.979,Z 740.516,A -85,B 0,C 180,E1 28339.786,E2 28339.786} C_VEL
LIN {X 0,Y 592.024,Z 730.153,A -85,B 0,C 180,E1 28338.209,E2 28338.209} C_VEL
LIN {X 0,Y 592.093,Z 718.354,A -85,B 0,C 180,E1 28336.724,E2 28336.724} C_VEL
LIN {X 0,Y 592.191,Z 704.588,A -85,B 0,C 180,E1 28335.28,E2 28335.28} C_VEL
LIN {X 0,Y 592.306,Z 689.606,A -85,B 0,C 180,E1 28333.979,E2 28333.979} C_VEL
LIN {X 0,Y 592.421,Z 673.433,A -85,B 0,C 180,E1 28332.822,E2 28332.822} C_VEL
LIN {X 0,Y 592.532,Z 657.052,A -85,B 0,C 180,E1 28331.861,E2 28331.861} C_VEL
LIN {X 0,Y 592.648,Z 640.128,A -85,B 0,C 180,E1 28331.062,E2 28331.062} C_VEL
LIN {X 0,Y 592.753,Z 621.869,A -85,B 0,C 180,E1 28330.397,E2 28330.397} C_VEL
LIN {X 0,Y 592.826,Z 603.348,A -85,B 0,C 180,E1 28329.912,E2 28329.912} C_VEL
LIN {X 0,Y 592.877,Z 583.633,A -85,B 0,C 180,E1 28329.587,E2 28329.587} C_VEL
LIN {X 0,Y 592.955,Z 387.8,A -85,B 0,C 180,E1 28327.09,E2 28327.09} C_VEL
LIN {X 0,Y 592.782,Z 385.95,A -85,B 0,C 180,E1 28327.022,E2 28327.022} C_VEL
LIN {X 0,Y 593.015,Z 340.267,A -85,B 0,C 180,E1 28323.952,E2 28323.952} C_VEL
LIN {X 0,Y 593.254,Z 297.56,A -85,B 0,C 180,E1 28321.011,E2 28321.011} C_VEL
LIN {X 0,Y 593.233,Z 280.972,A -85,B 0,C 180,E1 28319.841,E2 28319.841} C_VEL
LIN {X 0,Y 591.993,Z 277.059,A -85,B 0,C 180,E1 28319.472,E2 28319.472} C_VEL
LIN {X 0,Y 591.96,Z 277.057,A -85,B 0,C 180,E1 28316.554,E2 28316.554} C_VEL
LIN {X 0,Y 591.974,Z 277.056,A -85,B 0,C 180,E1 28313.28,E2 28313.28} C_VEL
LIN {X 0,Y 591.96,Z 277.056,A -85,B 0,C 180,E1 28310.449,E2 28310.449} C_VEL
LIN {X 0,Y 591.96,Z 277.056,A -85,B 0,C 180,E1 28307.104,E2 28307.104} C_VEL
LIN {X 0,Y 591.971,Z 277.056,A -85,B 0,C 180,E1 28304.264,E2 28304.264} C_VEL
LIN {X 0,Y 591.956,Z 277.055,A -85,B 0,C 180,E1 28300.975,E2 28300.975} C_VEL
LIN {X 0,Y 591.991,Z 277.055,A -85,B 0,C 180,E1 28298.06,E2 28298.06} C_VEL
LIN {X 0,Y 591.956,Z 277.055,A -85,B 0,C 180,E1 28294.932,E2 28294.932} C_VEL
LIN {X 0,Y 592.007,Z 277.055,A -85,B 0,C 180,E1 28291.914,E2 28291.914} C_VEL
LIN {X 0,Y 591.958,Z 277.055,A -85,B 0,C 180,E1 28288.887,E2 28288.887} C_VEL
LIN {X 0,Y 592.003,Z 277.055,A -85,B 0,C 180,E1 28285.941,E2 28285.941} C_VEL
LIN {X 0,Y 591.959,Z 277.054,A -85,B 0,C 180,E1 28282.861,E2 28282.861} C_VEL
LIN {X 0,Y 592.016,Z 277.055,A -85,B 0,C 180,E1 28279.83,E2 28279.83} C_VEL
LIN {X 0,Y 591.957,Z 277.054,A -85,B 0,C 180,E1 28276.688,E2 28276.688} C_VEL
LIN {X 0,Y 592.038,Z 277.054,A -85,B 0,C 180,E1 28273.578,E2 28273.578} C_VEL
LIN {X 0,Y 591.96,Z 277.054,A -85,B 0,C 180,E1 28270.512,E2 28270.512} C_VEL
LIN {X 0,Y 592.015,Z 277.053,A -85,B 0,C 180,E1 28267.376,E2 28267.376} C_VEL
LIN {X 0,Y 591.962,Z 277.054,A -85,B 0,C 180,E1 28264.457,E2 28264.457} C_VEL
LIN {X 0,Y 592.016,Z 277.053,A -85,B 0,C 180,E1 28261.356,E2 28261.356} C_VEL
LIN {X 0,Y 591.966,Z 277.054,A -85,B 0,C 180,E1 28258.356,E2 28258.356} C_VEL
LIN {X 0,Y 591.996,Z 277.053,A -85,B 0,C 180,E1 28255.157,E2 28255.157} C_VEL
LIN {X 0,Y 591.972,Z 277.054,A -85,B 0,C 180,E1 28252.236,E2 28252.236} C_VEL
LIN {X 0,Y 591.975,Z 277.054,A -85,B 0,C 180,E1 28250.18,E2 28250.18} C_VEL
LIN {X 0,Y 591.024,Z 277.179,A -85,B 0,C 180,E1 28249.435,E2 28249.435} C_VEL
LIN {X 0,Y 584.495,Z 277.99,A -85,B 0,C 180,E1 28247.288,E2 28247.288} C_VEL
LIN {X 0,Y 584.034,Z 278.042,A -85,B 0,C 180,E1 28246.798,E2 28246.798} C_VEL
LIN {X 0,Y 584.071,Z 278.044,A -85,B 0,C 180,E1 28243.799,E2 28243.799} C_VEL
LIN {X 0,Y 584.029,Z 278.042,A -85,B 0,C 180,E1 28240.604,E2 28240.604} C_VEL
LIN {X 0,Y 584.103,Z 278.041,A -85,B 0,C 180,E1 28237.455,E2 28237.455} C_VEL
LIN {X 0,Y 584.031,Z 278.042,A -85,B 0,C 180,E1 28234.336,E2 28234.336} C_VEL
LIN {X 0,Y 584.074,Z 278.04,A -85,B 0,C 180,E1 28231.137,E2 28231.137} C_VEL
LIN {X 0,Y 584.04,Z 278.043,A -85,B 0,C 180,E1 28228.116,E2 28228.116} C_VEL
LIN {X 0,Y 584.041,Z 278.041,A -85,B 0,C 180,E1 28224.745,E2 28224.745} C_VEL
LIN {X 0,Y 584.077,Z 278.044,A -85,B 0,C 180,E1 28221.709,E2 28221.709} C_VEL
LIN {X 0,Y 584.036,Z 278.041,A -85,B 0,C 180,E1 28218.509,E2 28218.509} C_VEL
LIN {X 0,Y 584.102,Z 278.042,A -85,B 0,C 180,E1 28215.405,E2 28215.405} C_VEL
LIN {X 0,Y 584.036,Z 278.042,A -85,B 0,C 180,E1 28212.283,E2 28212.283} C_VEL
LIN {X 0,Y 584.091,Z 278.039,A -85,B 0,C 180,E1 28209.158,E2 28209.158} C_VEL
LIN {X 0,Y 584.043,Z 278.042,A -85,B 0,C 180,E1 28206.079,E2 28206.079} C_VEL
LIN {X 0,Y 584.054,Z 278.04,A -85,B 0,C 180,E1 28202.749,E2 28202.749} C_VEL
LIN {X 0,Y 584.066,Z 278.043,A -85,B 0,C 180,E1 28199.764,E2 28199.764} C_VEL
LIN {X 0,Y 584.045,Z 278.04,A -85,B 0,C 180,E1 28196.539,E2 28196.539} C_VEL
LIN {X 0,Y 584.097,Z 278.043,A -85,B 0,C 180,E1 28193.398,E2 28193.398} C_VEL
LIN {X 0,Y 584.041,Z 278.041,A -85,B 0,C 180,E1 28190.231,E2 28190.231} C_VEL
LIN {X 0,Y 584.088,Z 278.038,A -85,B 0,C 180,E1 28187.02,E2 28187.02} C_VEL
LIN {X 0,Y 584.056,Z 278.042,A -85,B 0,C 180,E1 28183.866,E2 28183.866} C_VEL
LIN {X 0,Y 584.051,Z 278.039,A -85,B 0,C 180,E1 28180.554,E2 28180.554} C_VEL
LIN {X 0,Y 584.091,Z 278.044,A -85,B 0,C 180,E1 28177.474,E2 28177.474} C_VEL
LIN {X 0,Y 584.044,Z 278.04,A -85,B 0,C 180,E1 28174.319,E2 28174.319} C_VEL
LIN {X 0,Y 584.101,Z 278.04,A -85,B 0,C 180,E1 28171.176,E2 28171.176} C_VEL
LIN {X 0,Y 584.047,Z 278.041,A -85,B 0,C 180,E1 28168.037,E2 28168.037} C_VEL
LIN {X 0,Y 584.08,Z 278.037,A -85,B 0,C 180,E1 28164.794,E2 28164.794} C_VEL
LIN {X 0,Y 584.073,Z 278.043,A -85,B 0,C 180,E1 28161.633,E2 28161.633} C_VEL
LIN {X 0,Y 584.05,Z 278.039,A -85,B 0,C 180,E1 28158.345,E2 28158.345} C_VEL
LIN {X 0,Y 584.1,Z 278.041,A -85,B 0,C 180,E1 28155.222,E2 28155.222} C_VEL
LIN {X 0,Y 584.051,Z 278.04,A -85,B 0,C 180,E1 28152.052,E2 28152.052} C_VEL
LIN {X 0,Y 584.094,Z 278.036,A -85,B 0,C 180,E1 28148.826,E2 28148.826} C_VEL
LIN {X 0,Y 584.072,Z 278.043,A -85,B 0,C 180,E1 28145.598,E2 28145.598} C_VEL
LIN {X 0,Y 584.058,Z 278.038,A -85,B 0,C 180,E1 28142.358,E2 28142.358} C_VEL
LIN {X 0,Y 584.1,Z 278.042,A -85,B 0,C 180,E1 28139.214,E2 28139.214} C_VEL
LIN {X 0,Y 584.051,Z 278.04,A -85,B 0,C 180,E1 28136.075,E2 28136.075} C_VEL
LIN {X 0,Y 584.097,Z 278.036,A -85,B 0,C 180,E1 28132.823,E2 28132.823} C_VEL
LIN {X 0,Y 584.069,Z 278.042,A -85,B 0,C 180,E1 28129.618,E2 28129.618} C_VEL
LIN {X 0,Y 584.065,Z 278.038,A -85,B 0,C 180,E1 28126.378,E2 28126.378} C_VEL
LIN {X 0,Y 584.098,Z 278.042,A -85,B 0,C 180,E1 28123.178,E2 28123.178} C_VEL
LIN {X 0,Y 584.057,Z 278.04,A -85,B 0,C 180,E1 28120.064,E2 28120.064} C_VEL
LIN {X 0,Y 584.097,Z 278.039,A -85,B 0,C 180,E1 28116.925,E2 28116.925} C_VEL
LIN {X 0,Y 584.065,Z 278.042,A -85,B 0,C 180,E1 28113.684,E2 28113.684} C_VEL
LIN {X 0,Y 584.07,Z 278.039,A -85,B 0,C 180,E1 28110.329,E2 28110.329} C_VEL
LIN {X 0,Y 584.125,Z 278.244,A -85,B 0,C 180,E1 28107.163,E2 28107.163} C_VEL
LIN {X 0,Y 585.085,Z 283.423,A -85,B 0,C 180,E1 28106.541,E2 28106.541} C_VEL
LIN {X 0,Y 584.835,Z 311.573,A -85,B 0,C 180,E1 28103.419,E2 28103.419} C_VEL
LIN {X 0,Y 584.606,Z 342.287,A -85,B 0,C 180,E1 28100.105,E2 28100.105} C_VEL
LIN {X 0,Y 584.404,Z 373.489,A -85,B 0,C 180,E1 28096.805,E2 28096.805} C_VEL
LIN {X 0,Y 584.239,Z 404.938,A -85,B 0,C 180,E1 28093.549,E2 28093.549} C_VEL
LIN {X 0,Y 584.521,Z 418.174,A -85,B 0,C 180,E1 28093.378,E2 28093.378} C_VEL
LIN {X 0,Y 584.414,Z 516.476,A -85,B 0,C 180,E1 28092.14,E2 28092.14} C_VEL
LIN {X 0,Y 584.358,Z 531.237,A -85,B 0,C 180,E1 28091.774,E2 28091.774} C_VEL
LIN {X 0,Y 584.279,Z 546.127,A -85,B 0,C 180,E1 28091.198,E2 28091.198} C_VEL
LIN {X 0,Y 584.185,Z 559.174,A -85,B 0,C 180,E1 28090.501,E2 28090.501} C_VEL
LIN {X 0,Y 584.127,Z 571.876,A -85,B 0,C 180,E1 28089.614,E2 28089.614} C_VEL
LIN {X 0,Y 584.053,Z 583.538,A -85,B 0,C 180,E1 28088.564,E2 28088.564} C_VEL
LIN {X 0,Y 583.992,Z 593.784,A -85,B 0,C 180,E1 28087.376,E2 28087.376} C_VEL
LIN {X 0,Y 583.953,Z 601.765,A -85,B 0,C 180,E1 28086.191,E2 28086.191} C_VEL
LIN {X 0,Y 583.931,Z 608.852,A -85,B 0,C 180,E1 28084.811,E2 28084.811} C_VEL
LIN {X 0,Y 583.923,Z 614.169,A -85,B 0,C 180,E1 28083.336,E2 28083.336} C_VEL
LIN {X 0,Y 583.916,Z 617.303,A -85,B 0,C 180,E1 28081.961,E2 28081.961} C_VEL
LIN {X 0,Y 583.919,Z 618.881,A -85,B 0,C 180,E1 28080.489,E2 28080.489} C_VEL
LIN {X 0,Y 583.914,Z 618.549,A -85,B 0,C 180,E1 28078.919,E2 28078.919} C_VEL
LIN {X 0,Y 583.918,Z 616.348,A -85,B 0,C 180,E1 28077.447,E2 28077.447} C_VEL
LIN {X 0,Y 583.922,Z 612.597,A -85,B 0,C 180,E1 28076.071,E2 28076.071} C_VEL
LIN {X 0,Y 583.937,Z 606.521,A -85,B 0,C 180,E1 28074.595,E2 28074.595} C_VEL
LIN {X 0,Y 583.967,Z 598.854,A -85,B 0,C 180,E1 28073.253,E2 28073.253} C_VEL
LIN {X 0,Y 584.011,Z 590.556,A -85,B 0,C 180,E1 28072.127,E2 28072.127} C_VEL
LIN {X 0,Y 584.072,Z 580.276,A -85,B 0,C 180,E1 28071.026,E2 28071.026} C_VEL
LIN {X 0,Y 584.134,Z 568.572,A -85,B 0,C 180,E1 28070.043,E2 28070.043} C_VEL
LIN {X 0,Y 584.22,Z 556.103,A -85,B 0,C 180,E1 28069.227,E2 28069.227} C_VEL
LIN {X 0,Y 584.299,Z 542.465,A -85,B 0,C 180,E1 28068.55,E2 28068.55} C_VEL
LIN {X 0,Y 584.372,Z 527.996,A -85,B 0,C 180,E1 28068.041,E2 28068.041} C_VEL
LIN {X 0,Y 584.416,Z 513.257,A -85,B 0,C 180,E1 28067.713,E2 28067.713} C_VEL
LIN {X 0,Y 584.298,Z 405.416,A -85,B 0,C 180,E1 28066.369,E2 28066.369} C_VEL
LIN {X 0,Y 584.227,Z 404.561,A -85,B 0,C 180,E1 28066.338,E2 28066.338} C_VEL
LIN {X 0,Y 584.377,Z 372.762,A -85,B 0,C 180,E1 28063.028,E2 28063.028} C_VEL
LIN {X 0,Y 584.605,Z 342.982,A -85,B 0,C 180,E1 28059.879,E2 28059.879} C_VEL
LIN {X 0,Y 584.751,Z 314.551,A -85,B 0,C 180,E1 28056.813,E2 28056.813} C_VEL
LIN {X 0,Y 585.127,Z 286.852,A -85,B 0,C 180,E1 28053.731,E2 28053.731} C_VEL
LIN {X 0,Y 585.023,Z 281.799,A -85,B 0,C 180,E1 28053.145,E2 28053.145} C_VEL
LIN {X 0,Y 584.1,Z 278.044,A -85,B 0,C 180,E1 28052.637,E2 28052.637} C_VEL
LIN {X 0,Y 584.061,Z 278.044,A -85,B 0,C 180,E1 28049.439,E2 28049.439} C_VEL
LIN {X 0,Y 584.089,Z 278.037,A -85,B 0,C 180,E1 28046.196,E2 28046.196} C_VEL
LIN {X 0,Y 584.091,Z 278.042,A -85,B 0,C 180,E1 28042.913,E2 28042.913} C_VEL
LIN {X 0,Y 584.084,Z 278.041,A -85,B 0,C 180,E1 28039.678,E2 28039.678} C_VEL
LIN {X 0,Y 584.092,Z 278.036,A -85,B 0,C 180,E1 28036.38,E2 28036.38} C_VEL
LIN {X 0,Y 584.067,Z 278.042,A -85,B 0,C 180,E1 28033.083,E2 28033.083} C_VEL
LIN {X 0,Y 584.1,Z 278.042,A -85,B 0,C 180,E1 28029.924,E2 28029.924} C_VEL
LIN {X 0,Y 584.048,Z 278.042,A -85,B 0,C 180,E1 28026.812,E2 28026.812} C_VEL
LIN {X 0,Y 584.049,Z 278.047,A -85,B 0,C 180,E1 28023.517,E2 28023.517} C_VEL
LIN {X 0,Y 584.037,Z 278.116,A -85,B 0,C 180,E1 28020.876,E2 28020.876} C_VEL
LIN {X 0,Y 586.074,Z 284.425,A -85,B 0,C 180,E1 28020.316,E2 28020.316} C_VEL
LIN {X 0,Y 585.734,Z 325.908,A -85,B 0,C 180,E1 28017.396,E2 28017.396} C_VEL
LIN {X 0,Y 585.346,Z 371.807,A -85,B 0,C 180,E1 28014.247,E2 28014.247} C_VEL
LIN {X 0,Y 585.318,Z 387.181,A -85,B 0,C 180,E1 28013.234,E2 28013.234} C_VEL
LIN {X 0,Y 585.742,Z 393.105,A -85,B 0,C 180,E1 28013.139,E2 28013.139} C_VEL
LIN {X 0,Y 585.337,Z 596.286,A -85,B 0,C 180,E1 28010.499,E2 28010.499} C_VEL
LIN {X 0,Y 585.221,Z 615.284,A -85,B 0,C 180,E1 28010.064,E2 28010.064} C_VEL
LIN {X 0,Y 585.083,Z 633.387,A -85,B 0,C 180,E1 28009.466,E2 28009.466} C_VEL
LIN {X 0,Y 584.919,Z 651.037,A -85,B 0,C 180,E1 28008.695,E2 28008.695} C_VEL
LIN {X 0,Y 584.739,Z 668.222,A -85,B 0,C 180,E1 28007.744,E2 28007.744} C_VEL
LIN {X 0,Y 584.561,Z 684.227,A -85,B 0,C 180,E1 28006.654,E2 28006.654} C_VEL
LIN {X 0,Y 584.393,Z 699.1,A -85,B 0,C 180,E1 28005.431,E2 28005.431} C_VEL
LIN {X 0,Y 584.241,Z 712.939,A -85,B 0,C 180,E1 28004.065,E2 28004.065} C_VEL
LIN {X 0,Y 584.125,Z 725.679,A -85,B 0,C 180,E1 28002.556,E2 28002.556} C_VEL
LIN {X 0,Y 584.042,Z 736.862,A -85,B 0,C 180,E1 28000.955,E2 28000.955} C_VEL
LIN {X 0,Y 583.979,Z 746.506,A -85,B 0,C 180,E1 27999.262,E2 27999.262} C_VEL
LIN {X 0,Y 583.944,Z 754.4,A -85,B 0,C 180,E1 27997.522,E2 27997.522} C_VEL
LIN {X 0,Y 583.917,Z 760.409,A -85,B 0,C 180,E1 27995.799,E2 27995.799} C_VEL
LIN {X 0,Y 583.917,Z 764.873,A -85,B 0,C 180,E1 27994.027,E2 27994.027} C_VEL
LIN {X 0,Y 583.911,Z 767.789,A -85,B 0,C 180,E1 27992.16,E2 27992.16} C_VEL
LIN {X 0,Y 583.908,Z 768.939,A -85,B 0,C 180,E1 27990.295,E2 27990.295} C_VEL
LIN {X 0,Y 583.913,Z 768.349,A -85,B 0,C 180,E1 27988.431,E2 27988.431} C_VEL
LIN {X 0,Y 583.907,Z 766.007,A -85,B 0,C 180,E1 27986.565,E2 27986.565} C_VEL
LIN {X 0,Y 583.923,Z 762.1,A -85,B 0,C 180,E1 27984.794,E2 27984.794} C_VEL
LIN {X 0,Y 583.937,Z 756.47,A -85,B 0,C 180,E1 27983.018,E2 27983.018} C_VEL
LIN {X 0,Y 583.956,Z 749.429,A -85,B 0,C 180,E1 27981.335,E2 27981.335} C_VEL
LIN {X 0,Y 584.016,Z 740.517,A -85,B 0,C 180,E1 27979.645,E2 27979.645} C_VEL
LIN {X 0,Y 584.086,Z 730.154,A -85,B 0,C 180,E1 27978.047,E2 27978.047} C_VEL
LIN {X 0,Y 584.195,Z 718.355,A -85,B 0,C 180,E1 27976.541,E2 27976.541} C_VEL
LIN {X 0,Y 584.341,Z 704.587,A -85,B 0,C 180,E1 27975.078,E2 27975.078} C_VEL
LIN {X 0,Y 584.507,Z 689.608,A -85,B 0,C 180,E1 27973.76,E2 27973.76} C_VEL
LIN {X 0,Y 584.686,Z 673.436,A -85,B 0,C 180,E1 27972.587,E2 27972.587} C_VEL
LIN {X 0,Y 584.862,Z 656.537,A -85,B 0,C 180,E1 27971.588,E2 27971.588} C_VEL
LIN {X 0,Y 585.031,Z 639.819,A -85,B 0,C 180,E1 27970.793,E2 27970.793} C_VEL
LIN {X 0,Y 585.189,Z 621.656,A -85,B 0,C 180,E1 27970.126,E2 27970.126} C_VEL
LIN {X 0,Y 585.303,Z 603.186,A -85,B 0,C 180,E1 27969.639,E2 27969.639} C_VEL
LIN {X 0,Y 585.38,Z 583.224,A -85,B 0,C 180,E1 27969.309,E2 27969.309} C_VEL
LIN {X 0,Y 585.576,Z 388.814,A -85,B 0,C 180,E1 27966.798,E2 27966.798} C_VEL
LIN {X 0,Y 585.243,Z 386.265,A -85,B 0,C 180,E1 27966.73,E2 27966.73} C_VEL
LIN {X 0,Y 585.607,Z 340.189,A -85,B 0,C 180,E1 27963.592,E2 27963.592} C_VEL
LIN {X 0,Y 585.963,Z 297.656,A -85,B 0,C 180,E1 27960.623,E2 27960.623} C_VEL
LIN {X 0,Y 585.915,Z 283.558,A -85,B 0,C 180,E1 27959.614,E2 27959.614} C_VEL
LIN {X 0,Y 584.023,Z 278.049,A -85,B 0,C 180,E1 27959.097,E2 27959.097} C_VEL
LIN {X 0,Y 584.054,Z 278.046,A -85,B 0,C 180,E1 27956.129,E2 27956.129} C_VEL
LIN {X 0,Y 584.015,Z 278.045,A -85,B 0,C 180,E1 27952.942,E2 27952.942} C_VEL
LIN {X 0,Y 584.075,Z 278.045,A -85,B 0,C 180,E1 27949.926,E2 27949.926} C_VEL
LIN {X 0,Y 584.012,Z 278.045,A -85,B 0,C 180,E1 27946.831,E2 27946.831} C_VEL
LIN {X 0,Y 584.092,Z 278.045,A -85,B 0,C 180,E1 27943.75,E2 27943.75} C_VEL
LIN {X 0,Y 584.012,Z 278.045,A -85,B 0,C 180,E1 27940.675,E2 27940.675} C_VEL
LIN {X 0,Y 584.074,Z 278.044,A -85,B 0,C 180,E1 27937.549,E2 27937.549} C_VEL
LIN {X 0,Y 584.016,Z 278.044,A -85,B 0,C 180,E1 27934.566,E2 27934.566} C_VEL
LIN {X 0,Y 584.053,Z 278.044,A -85,B 0,C 180,E1 27931.362,E2 27931.362} C_VEL
LIN {X 0,Y 584.022,Z 278.044,A -85,B 0,C 180,E1 27928.422,E2 27928.422} C_VEL
LIN {X 0,Y 584.033,Z 278.043,A -85,B 0,C 180,E1 27925.092,E2 27925.092} C_VEL
LIN {X 0,Y 584.034,Z 278.044,A -85,B 0,C 180,E1 27922.232,E2 27922.232} C_VEL
LIN {X 0,Y 584.028,Z 278.043,A -85,B 0,C 180,E1 27918.984,E2 27918.984} C_VEL
LIN {X 0,Y 584.044,Z 278.044,A -85,B 0,C 180,E1 27916.102,E2 27916.102} C_VEL
LIN {X 0,Y 584.024,Z 278.043,A -85,B 0,C 180,E1 27912.861,E2 27912.861} C_VEL
LIN {X 0,Y 584.071,Z 278.044,A -85,B 0,C 180,E1 27909.858,E2 27909.858} C_VEL
LIN {X 0,Y 584.022,Z 278.043,A -85,B 0,C 180,E1 27906.687,E2 27906.687} C_VEL
LIN {X 0,Y 584.096,Z 278.042,A -85,B 0,C 180,E1 27903.534,E2 27903.534} C_VEL
LIN {X 0,Y 584.024,Z 278.043,A -85,B 0,C 180,E1 27900.492,E2 27900.492} C_VEL
LIN {X 0,Y 584.08,Z 278.041,A -85,B 0,C 180,E1 27897.352,E2 27897.352} C_VEL
LIN {X 0,Y 584.03,Z 278.043,A -85,B 0,C 180,E1 27894.303,E2 27894.303} C_VEL
LIN {X 0,Y 584.048,Z 278.042,A -85,B 0,C 180,E1 27891.032,E2 27891.032} C_VEL
LIN {X 0,Y 584.046,Z 278.043,A -85,B 0,C 180,E1 27888.047,E2 27888.047} C_VEL
LIN {X 0,Y 584.034,Z 278.042,A -85,B 0,C 180,E1 27886.798,E2 27886.798} C_VEL
LIN {X 0,Y 583.038,Z 278.169,A -85,B 0,C 180,E1 27886.042,E2 27886.042} C_VEL
LIN {X 0,Y 576.61,Z 278.979,A -85,B 0,C 180,E1 27883.866,E2 27883.866} C_VEL
LIN {X 0,Y 576.152,Z 279.03,A -85,B 0,C 180,E1 27883.369,E2 27883.369} C_VEL
LIN {X 0,Y 576.093,Z 279.031,A -85,B 0,C 180,E1 27880.326,E2 27880.326} C_VEL
LIN {X 0,Y 576.127,Z 279.03,A -85,B 0,C 180,E1 27877.125,E2 27877.125} C_VEL
LIN {X 0,Y 576.105,Z 279.032,A -85,B 0,C 180,E1 27874.067,E2 27874.067} C_VEL
LIN {X 0,Y 576.104,Z 279.03,A -85,B 0,C 180,E1 27870.805,E2 27870.805} C_VEL
LIN {X 0,Y 576.128,Z 279.032,A -85,B 0,C 180,E1 27867.808,E2 27867.808} C_VEL
LIN {X 0,Y 576.096,Z 279.03,A -85,B 0,C 180,E1 27864.574,E2 27864.574} C_VEL
LIN {X 0,Y 576.162,Z 279.031,A -85,B 0,C 180,E1 27861.467,E2 27861.467} C_VEL
LIN {X 0,Y 576.097,Z 279.031,A -85,B 0,C 180,E1 27858.269,E2 27858.269} C_VEL
LIN {X 0,Y 576.138,Z 279.028,A -85,B 0,C 180,E1 27855.066,E2 27855.066} C_VEL
LIN {X 0,Y 576.107,Z 279.031,A -85,B 0,C 180,E1 27852.032,E2 27852.032} C_VEL
LIN {X 0,Y 576.106,Z 279.029,A -85,B 0,C 180,E1 27848.652,E2 27848.652} C_VEL
LIN {X 0,Y 576.151,Z 279.034,A -85,B 0,C 180,E1 27845.525,E2 27845.525} C_VEL
LIN {X 0,Y 576.101,Z 279.03,A -85,B 0,C 180,E1 27842.309,E2 27842.309} C_VEL
LIN {X 0,Y 576.16,Z 279.028,A -85,B 0,C 180,E1 27839.185,E2 27839.185} C_VEL
LIN {X 0,Y 576.107,Z 279.031,A -85,B 0,C 180,E1 27836.045,E2 27836.045} C_VEL
LIN {X 0,Y 576.114,Z 279.028,A -85,B 0,C 180,E1 27832.661,E2 27832.661} C_VEL
LIN {X 0,Y 576.146,Z 279.033,A -85,B 0,C 180,E1 27829.56,E2 27829.56} C_VEL
LIN {X 0,Y 576.104,Z 279.029,A -85,B 0,C 180,E1 27826.319,E2 27826.319} C_VEL
LIN {X 0,Y 576.16,Z 279.028,A -85,B 0,C 180,E1 27823.139,E2 27823.139} C_VEL
LIN {X 0,Y 576.11,Z 279.031,A -85,B 0,C 180,E1 27819.994,E2 27819.994} C_VEL
LIN {X 0,Y 576.124,Z 279.027,A -85,B 0,C 180,E1 27816.677,E2 27816.677} C_VEL
LIN {X 0,Y 576.151,Z 279.033,A -85,B 0,C 180,E1 27813.481,E2 27813.481} C_VEL
LIN {X 0,Y 576.107,Z 279.029,A -85,B 0,C 180,E1 27810.298,E2 27810.298} C_VEL
LIN {X 0,Y 576.162,Z 279.028,A -85,B 0,C 180,E1 27807.115,E2 27807.115} C_VEL
LIN {X 0,Y 576.114,Z 279.03,A -85,B 0,C 180,E1 27803.922,E2 27803.922} C_VEL
LIN {X 0,Y 576.126,Z 279.027,A -85,B 0,C 180,E1 27800.61,E2 27800.61} C_VEL
LIN {X 0,Y 576.149,Z 279.033,A -85,B 0,C 180,E1 27797.471,E2 27797.471} C_VEL
LIN {X 0,Y 576.112,Z 279.028,A -85,B 0,C 180,E1 27794.291,E2 27794.291} C_VEL
LIN {X 0,Y 576.16,Z 279.028,A -85,B 0,C 180,E1 27791.063,E2 27791.063} C_VEL
LIN {X 0,Y 576.116,Z 279.03,A -85,B 0,C 180,E1 27787.876,E2 27787.876} C_VEL
LIN {X 0,Y 576.135,Z 279.026,A -85,B 0,C 180,E1 27784.617,E2 27784.617} C_VEL
LIN {X 0,Y 576.154,Z 279.033,A -85,B 0,C 180,E1 27781.381,E2 27781.381} C_VEL
LIN {X 0,Y 576.114,Z 279.028,A -85,B 0,C 180,E1 27778.156,E2 27778.156} C_VEL
LIN {X 0,Y 576.158,Z 279.027,A -85,B 0,C 180,E1 27774.941,E2 27774.941} C_VEL
LIN {X 0,Y 576.125,Z 279.031,A -85,B 0,C 180,E1 27771.715,E2 27771.715} C_VEL
LIN {X 0,Y 576.123,Z 279.027,A -85,B 0,C 180,E1 27768.34,E2 27768.34} C_VEL
LIN {X 0,Y 576.16,Z 279.032,A -85,B 0,C 180,E1 27765.205,E2 27765.205} C_VEL
LIN {X 0,Y 576.117,Z 279.028,A -85,B 0,C 180,E1 27762.029,E2 27762.029} C_VEL
LIN {X 0,Y 576.162,Z 279.026,A -85,B 0,C 180,E1 27758.787,E2 27758.787} C_VEL
LIN {X 0,Y 576.138,Z 279.032,A -85,B 0,C 180,E1 27755.518,E2 27755.518} C_VEL
LIN {X 0,Y 576.122,Z 279.027,A -85,B 0,C 180,E1 27752.192,E2 27752.192} C_VEL
LIN {X 0,Y 576.159,Z 279.033,A -85,B 0,C 180,E1 27748.956,E2 27748.956} C_VEL
LIN {X 0,Y 576.156,Z 279.159,A -85,B 0,C 180,E1 27747.468,E2 27747.468} C_VEL
LIN {X 0,Y 577.495,Z 285.407,A -85,B 0,C 180,E1 27746.697,E2 27746.697} C_VEL
LIN {X 0,Y 577.16,Z 313.584,A -85,B 0,C 180,E1 27743.533,E2 27743.533} C_VEL
LIN {X 0,Y 576.84,Z 343.755,A -85,B 0,C 180,E1 27740.229,E2 27740.229} C_VEL
LIN {X 0,Y 576.568,Z 374.958,A -85,B 0,C 180,E1 27736.884,E2 27736.884} C_VEL
LIN {X 0,Y 576.359,Z 404.948,A -85,B 0,C 180,E1 27733.738,E2 27733.738} C_VEL
LIN {X 0,Y 576.746,Z 412.628,A -85,B 0,C 180,E1 27733.632,E2 27733.632} C_VEL
LIN {X 0,Y 576.59,Z 516.436,A -85,B 0,C 180,E1 27732.309,E2 27732.309} C_VEL
LIN {X 0,Y 576.517,Z 531.333,A -85,B 0,C 180,E1 27731.934,E2 27731.934} C_VEL
LIN {X 0,Y 576.411,Z 546.143,A -85,B 0,C 180,E1 27731.353,E2 27731.353} C_VEL
LIN {X 0,Y 576.291,Z 559.182,A -85,B 0,C 180,E1 27730.646,E2 27730.646} C_VEL
LIN {X 0,Y 576.205,Z 571.373,A -85,B 0,C 180,E1 27729.789,E2 27729.789} C_VEL
LIN {X 0,Y 576.101,Z 583.544,A -85,B 0,C 180,E1 27728.683,E2 27728.683} C_VEL
LIN {X 0,Y 576.019,Z 593.789,A -85,B 0,C 180,E1 27727.479,E2 27727.479} C_VEL
LIN {X 0,Y 575.968,Z 601.769,A -85,B 0,C 180,E1 27726.277,E2 27726.277} C_VEL
LIN {X 0,Y 575.936,Z 608.854,A -85,B 0,C 180,E1 27724.878,E2 27724.878} C_VEL
LIN {X 0,Y 575.924,Z 614.183,A -85,B 0,C 180,E1 27723.379,E2 27723.379} C_VEL
LIN {X 0,Y 575.916,Z 617.462,A -85,B 0,C 180,E1 27721.889,E2 27721.889} C_VEL
LIN {X 0,Y 575.918,Z 618.907,A -85,B 0,C 180,E1 27720.396,E2 27720.396} C_VEL
LIN {X 0,Y 575.914,Z 618.548,A -85,B 0,C 180,E1 27718.904,E2 27718.904} C_VEL
LIN {X 0,Y 575.918,Z 616.347,A -85,B 0,C 180,E1 27717.411,E2 27717.411} C_VEL
LIN {X 0,Y 575.924,Z 612.595,A -85,B 0,C 180,E1 27716.017,E2 27716.017} C_VEL
LIN {X 0,Y 575.945,Z 606.518,A -85,B 0,C 180,E1 27714.52,E2 27714.52} C_VEL
LIN {X 0,Y 575.984,Z 599.066,A -85,B 0,C 180,E1 27713.193,E2 27713.193} C_VEL
LIN {X 0,Y 576.044,Z 590.551,A -85,B 0,C 180,E1 27712.017,E2 27712.017} C_VEL
LIN {X 0,Y 576.132,Z 579.868,A -85,B 0,C 180,E1 27710.862,E2 27710.862} C_VEL
LIN {X 0,Y 576.217,Z 568.222,A -85,B 0,C 180,E1 27709.88,E2 27709.88} C_VEL
LIN {X 0,Y 576.336,Z 555.661,A -85,B 0,C 180,E1 27709.053,E2 27709.053} C_VEL
LIN {X 0,Y 576.439,Z 542.449,A -85,B 0,C 180,E1 27708.391,E2 27708.391} C_VEL
LIN {X 0,Y 576.535,Z 527.974,A -85,B 0,C 180,E1 27707.876,E2 27707.876} C_VEL
LIN {X 0,Y 576.597,Z 513.214,A -85,B 0,C 180,E1 27707.544,E2 27707.544} C_VEL
LIN {X 0,Y 576.511,Z 406.048,A -85,B 0,C 180,E1 27706.189,E2 27706.189} C_VEL
LIN {X 0,Y 576.348,Z 404.554,A -85,B 0,C 180,E1 27706.147,E2 27706.147} C_VEL
LIN {X 0,Y 576.548,Z 372.849,A -85,B 0,C 180,E1 27702.8,E2 27702.8} C_VEL
LIN {X 0,Y 576.843,Z 343.094,A -85,B 0,C 180,E1 27699.61,E2 27699.61} C_VEL
LIN {X 0,Y 577.11,Z 314.948,A -85,B 0,C 180,E1 27696.516,E2 27696.516} C_VEL
LIN {X 0,Y 577.685,Z 285.53,A -85,B 0,C 180,E1 27693.144,E2 27693.144} C_VEL
LIN {X 0,Y 576.155,Z 279.031,A -85,B 0,C 180,E1 27692.283,E2 27692.283} C_VEL
LIN {X 0,Y 576.153,Z 279.034,A -85,B 0,C 180,E1 27688.974,E2 27688.974} C_VEL
LIN {X 0,Y 576.13,Z 279.03,A -85,B 0,C 180,E1 27685.664,E2 27685.664} C_VEL
LIN {X 0,Y 576.154,Z 279.026,A -85,B 0,C 180,E1 27682.473,E2 27682.473} C_VEL
LIN {X 0,Y 576.151,Z 279.033,A -85,B 0,C 180,E1 27679.136,E2 27679.136} C_VEL
LIN {X 0,Y 576.152,Z 279.029,A -85,B 0,C 180,E1 27675.9,E2 27675.9} C_VEL
LIN {X 0,Y 576.127,Z 279.029,A -85,B 0,C 180,E1 27672.733,E2 27672.733} C_VEL
LIN {X 0,Y 576.132,Z 279.033,A -85,B 0,C 180,E1 27669.434,E2 27669.434} C_VEL
LIN {X 0,Y 576.156,Z 279.03,A -85,B 0,C 180,E1 27666.2,E2 27666.2} C_VEL
LIN {X 0,Y 576.092,Z 279.036,A -85,B 0,C 180,E1 27663.024,E2 27663.024} C_VEL
LIN {X 0,Y 576.1,Z 279.144,A -85,B 0,C 180,E1 27661.229,E2 27661.229} C_VEL
LIN {X 0,Y 578.74,Z 286.962,A -85,B 0,C 180,E1 27660.527,E2 27660.527} C_VEL
LIN {X 0,Y 578.384,Z 326.448,A -85,B 0,C 180,E1 27657.736,E2 27657.736} C_VEL
LIN {X 0,Y 577.858,Z 372.458,A -85,B 0,C 180,E1 27654.537,E2 27654.537} C_VEL
LIN {X 0,Y 577.796,Z 387.181,A -85,B 0,C 180,E1 27653.555,E2 27653.555} C_VEL
LIN {X 0,Y 578.383,Z 393.359,A -85,B 0,C 180,E1 27653.448,E2 27653.448} C_VEL
LIN {X 0,Y 577.841,Z 596.286,A -85,B 0,C 180,E1 27650.777,E2 27650.777} C_VEL
LIN {X 0,Y 577.687,Z 615.283,A -85,B 0,C 180,E1 27650.337,E2 27650.337} C_VEL
LIN {X 0,Y 577.5,Z 633.385,A -85,B 0,C 180,E1 27649.732,E2 27649.732} C_VEL
LIN {X 0,Y 577.273,Z 651.33,A -85,B 0,C 180,E1 27648.936,E2 27648.936} C_VEL
LIN {X 0,Y 577.028,Z 668.579,A -85,B 0,C 180,E1 27647.966,E2 27647.966} C_VEL
LIN {X 0,Y 576.782,Z 684.959,A -85,B 0,C 180,E1 27646.829,E2 27646.829} C_VEL
LIN {X 0,Y 576.551,Z 700.217,A -85,B 0,C 180,E1 27645.542,E2 27645.542} C_VEL
LIN {X 0,Y 576.349,Z 714.174,A -85,B 0,C 180,E1 27644.125,E2 27644.125} C_VEL
LIN {X 0,Y 576.197,Z 726.453,A -85,B 0,C 180,E1 27642.63,E2 27642.63} C_VEL
LIN {X 0,Y 576.084,Z 737.498,A -85,B 0,C 180,E1 27641.007,E2 27641.007} C_VEL
LIN {X 0,Y 576.001,Z 747.02,A -85,B 0,C 180,E1 27639.291,E2 27639.291} C_VEL
LIN {X 0,Y 575.956,Z 754.58,A -85,B 0,C 180,E1 27637.582,E2 27637.582} C_VEL
LIN {X 0,Y 575.92,Z 760.711,A -85,B 0,C 180,E1 27635.78,E2 27635.78} C_VEL
LIN {X 0,Y 575.919,Z 765.078,A -85,B 0,C 180,E1 27633.983,E2 27633.983} C_VEL
LIN {X 0,Y 575.912,Z 767.901,A -85,B 0,C 180,E1 27632.09,E2 27632.09} C_VEL
LIN {X 0,Y 575.91,Z 768.962,A -85,B 0,C 180,E1 27630.2,E2 27630.2} C_VEL
LIN {X 0,Y 575.91,Z 768.281,A -85,B 0,C 180,E1 27628.309,E2 27628.309} C_VEL
LIN {X 0,Y 575.911,Z 765.846,A -85,B 0,C 180,E1 27626.417,E2 27626.417} C_VEL
LIN {X 0,Y 575.923,Z 761.592,A -85,B 0,C 180,E1 27624.522,E2 27624.522} C_VEL
LIN {X 0,Y 575.951,Z 755.395,A -85,B 0,C 180,E1 27622.62,E2 27622.62} C_VEL
LIN {X 0,Y 576.003,Z 747.542,A -85,B 0,C 180,E1 27620.811,E2 27620.811} C_VEL
LIN {X 0,Y 576.076,Z 738.143,A -85,B 0,C 180,E1 27619.096,E2 27619.096} C_VEL
LIN {X 0,Y 576.192,Z 727.235,A -85,B 0,C 180,E1 27617.473,E2 27617.473} C_VEL
LIN {X 0,Y 576.344,Z 714.806,A -85,B 0,C 180,E1 27615.944,E2 27615.944} C_VEL
LIN {X 0,Y 576.541,Z 700.784,A -85,B 0,C 180,E1 27614.511,E2 27614.511} C_VEL
LIN {X 0,Y 576.769,Z 685.645,A -85,B 0,C 180,E1 27613.225,E2 27613.225} C_VEL
LIN {X 0,Y 577.012,Z 669.413,A -85,B 0,C 180,E1 27612.088,E2 27612.088} C_VEL
LIN {X 0,Y 577.238,Z 653.071,A -85,B 0,C 180,E1 27611.154,E2 27611.154} C_VEL
LIN {X 0,Y 577.455,Z 635.99,A -85,B 0,C 180,E1 27610.373,E2 27610.373} C_VEL
LIN {X 0,Y 577.654,Z 617.313,A -85,B 0,C 180,E1 27609.723,E2 27609.723} C_VEL
LIN {X 0,Y 577.812,Z 598.64,A -85,B 0,C 180,E1 27609.27,E2 27609.27} C_VEL
LIN {X 0,Y 577.928,Z 569.05,A -85,B 0,C 180,E1 27608.845,E2 27608.845} C_VEL
LIN {X 0,Y 578.223,Z 389.896,A -85,B 0,C 180,E1 27606.499,E2 27606.499} C_VEL
LIN {X 0,Y 577.724,Z 386.265,A -85,B 0,C 180,E1 27606.409,E2 27606.409} C_VEL
LIN {X 0,Y 578.234,Z 339.401,A -85,B 0,C 180,E1 27603.173,E2 27603.173} C_VEL
LIN {X 0,Y 578.667,Z 297.5,A -85,B 0,C 180,E1 27600.215,E2 27600.215} C_VEL
LIN {X 0,Y 578.652,Z 286.636,A -85,B 0,C 180,E1 27599.434,E2 27599.434} C_VEL
LIN {X 0,Y 576.078,Z 279.039,A -85,B 0,C 180,E1 27598.71,E2 27598.71} C_VEL
LIN {X 0,Y 576.123,Z 279.035,A -85,B 0,C 180,E1 27595.524,E2 27595.524} C_VEL
LIN {X 0,Y 576.083,Z 279.034,A -85,B 0,C 180,E1 27592.469,E2 27592.469} C_VEL
LIN {X 0,Y 576.085,Z 279.034,A -85,B 0,C 180,E1 27589.133,E2 27589.133} C_VEL
LIN {X 0,Y 576.103,Z 279.034,A -85,B 0,C 180,E1 27586.174,E2 27586.174} C_VEL
LIN {X 0,Y 576.077,Z 279.033,A -85,B 0,C 180,E1 27582.91,E2 27582.91} C_VEL
LIN {X 0,Y 576.154,Z 279.034,A -85,B 0,C 180,E1 27579.757,E2 27579.757} C_VEL
LIN {X 0,Y 576.074,Z 279.033,A -85,B 0,C 180,E1 27576.661,E2 27576.661} C_VEL
LIN {X 0,Y 576.132,Z 279.032,A -85,B 0,C 180,E1 27573.497,E2 27573.497} C_VEL
LIN {X 0,Y 576.081,Z 279.033,A -85,B 0,C 180,E1 27570.452,E2 27570.452} C_VEL
LIN {X 0,Y 576.097,Z 279.032,A -85,B 0,C 180,E1 27567.16,E2 27567.16} C_VEL
LIN {X 0,Y 576.099,Z 279.033,A -85,B 0,C 180,E1 27564.18,E2 27564.18} C_VEL
LIN {X 0,Y 576.087,Z 279.032,A -85,B 0,C 180,E1 27560.95,E2 27560.95} C_VEL
LIN {X 0,Y 576.129,Z 279.033,A -85,B 0,C 180,E1 27557.89,E2 27557.89} C_VEL
LIN {X 0,Y 576.083,Z 279.032,A -85,B 0,C 180,E1 27554.783,E2 27554.783} C_VEL
LIN {X 0,Y 576.151,Z 279.033,A -85,B 0,C 180,E1 27551.716,E2 27551.716} C_VEL
LIN {X 0,Y 576.082,Z 279.032,A -85,B 0,C 180,E1 27548.585,E2 27548.585} C_VEL
LIN {X 0,Y 576.15,Z 279.031,A -85,B 0,C 180,E1 27545.478,E2 27545.478} C_VEL
LIN {X 0,Y 576.087,Z 279.032,A -85,B 0,C 180,E1 27542.389,E2 27542.389} C_VEL
LIN {X 0,Y 576.111,Z 279.031,A -85,B 0,C 180,E1 27539.106,E2 27539.106} C_VEL
LIN {X 0,Y 576.102,Z 279.032,A -85,B 0,C 180,E1 27536.12,E2 27536.12} C_VEL
LIN {X 0,Y 576.094,Z 279.031,A -85,B 0,C 180,E1 27532.823,E2 27532.823} C_VEL
LIN {X 0,Y 576.134,Z 279.033,A -85,B 0,C 180,E1 27529.806,E2 27529.806} C_VEL
LIN {X 0,Y 576.09,Z 279.031,A -85,B 0,C 180,E1 27526.656,E2 27526.656} C_VEL
LIN {X 0,Y 576.158,Z 279.033,A -85,B 0,C 180,E1 27523.57,E2 27523.57} C_VEL
LIN {X 0,Y 576.152,Z 279.03,A -85,B 0,C 180,E1 27523.369,E2 27523.369} C_VEL
LIN {X 0,Y 575.111,Z 279.157,A -85,B 0,C 180,E1 27522.603,E2 27522.603} C_VEL
LIN {X 0,Y 568.667,Z 279.958,A -85,B 0,C 180,E1 27520.454,E2 27520.454} C_VEL
LIN {X 0,Y 568.182,Z 280.021,A -85,B 0,C 180,E1 27519.894,E2 27519.894} C_VEL
LIN {X 0,Y 568.155,Z 280.02,A -85,B 0,C 180,E1 27516.676,E2 27516.676} C_VEL
LIN {X 0,Y 568.216,Z 280.023,A -85,B 0,C 180,E1 27513.567,E2 27513.567} C_VEL
LIN {X 0,Y 568.155,Z 280.02,A -85,B 0,C 180,E1 27510.365,E2 27510.365} C_VEL
LIN {X 0,Y 568.203,Z 280.018,A -85,B 0,C 180,E1 27507.184,E2 27507.184} C_VEL
LIN {X 0,Y 568.168,Z 280.021,A -85,B 0,C 180,E1 27504.046,E2 27504.046} C_VEL
LIN {X 0,Y 568.162,Z 280.019,A -85,B 0,C 180,E1 27500.692,E2 27500.692} C_VEL
LIN {X 0,Y 568.205,Z 280.022,A -85,B 0,C 180,E1 27497.63,E2 27497.63} C_VEL
LIN {X 0,Y 568.159,Z 280.019,A -85,B 0,C 180,E1 27494.402,E2 27494.402} C_VEL
LIN {X 0,Y 568.211,Z 280.017,A -85,B 0,C 180,E1 27491.155,E2 27491.155} C_VEL
LIN {X 0,Y 568.169,Z 280.02,A -85,B 0,C 180,E1 27488.018,E2 27488.018} C_VEL
LIN {X 0,Y 568.168,Z 280.018,A -85,B 0,C 180,E1 27484.639,E2 27484.639} C_VEL
LIN {X 0,Y 568.216,Z 280.022,A -85,B 0,C 180,E1 27481.507,E2 27481.507} C_VEL
LIN {X 0,Y 568.162,Z 280.019,A -85,B 0,C 180,E1 27478.368,E2 27478.368} C_VEL
LIN {X 0,Y 568.221,Z 280.017,A -85,B 0,C 180,E1 27475.202,E2 27475.202} C_VEL
LIN {X 0,Y 568.172,Z 280.02,A -85,B 0,C 180,E1 27471.973,E2 27471.973} C_VEL
LIN {X 0,Y 568.171,Z 280.018,A -85,B 0,C 180,E1 27468.573,E2 27468.573} C_VEL
LIN {X 0,Y 568.222,Z 280.02,A -85,B 0,C 180,E1 27465.371,E2 27465.371} C_VEL
LIN {X 0,Y 568.166,Z 280.019,A -85,B 0,C 180,E1 27462.19,E2 27462.19} C_VEL
LIN {X 0,Y 568.203,Z 280.016,A -85,B 0,C 180,E1 27458.907,E2 27458.907} C_VEL
LIN {X 0,Y 568.186,Z 280.02,A -85,B 0,C 180,E1 27455.756,E2 27455.756} C_VEL
LIN {X 0,Y 568.171,Z 280.018,A -85,B 0,C 180,E1 27452.42,E2 27452.42} C_VEL
LIN {X 0,Y 568.223,Z 280.018,A -85,B 0,C 180,E1 27449.193,E2 27449.193} C_VEL
LIN {X 0,Y 568.173,Z 280.019,A -85,B 0,C 180,E1 27445.963,E2 27445.963} C_VEL
LIN {X 0,Y 568.188,Z 280.016,A -85,B 0,C 180,E1 27442.619,E2 27442.619} C_VEL
LIN {X 0,Y 568.211,Z 280.022,A -85,B 0,C 180,E1 27439.454,E2 27439.454} C_VEL
LIN {X 0,Y 568.171,Z 280.018,A -85,B 0,C 180,E1 27436.253,E2 27436.253} C_VEL
LIN {X 0,Y 568.221,Z 280.016,A -85,B 0,C 180,E1 27433.016,E2 27433.016} C_VEL
LIN {X 0,Y 568.181,Z 280.019,A -85,B 0,C 180,E1 27429.823,E2 27429.823} C_VEL
LIN {X 0,Y 568.184,Z 280.016,A -85,B 0,C 180,E1 27426.455,E2 27426.455} C_VEL
LIN {X 0,Y 568.222,Z 280.02,A -85,B 0,C 180,E1 27423.226,E2 27423.226} C_VEL
LIN {X 0,Y 568.176,Z 280.018,A -85,B 0,C 180,E1 27419.97,E2 27419.97} C_VEL
LIN {X 0,Y 568.208,Z 280.014,A -85,B 0,C 180,E1 27416.699,E2 27416.699} C_VEL
LIN {X 0,Y 568.215,Z 280.022,A -85,B 0,C 180,E1 27413.378,E2 27413.378} C_VEL
LIN {X 0,Y 568.177,Z 280.017,A -85,B 0,C 180,E1 27410.104,E2 27410.104} C_VEL
LIN {X 0,Y 568.22,Z 280.015,A -85,B 0,C 180,E1 27406.904,E2 27406.904} C_VEL
LIN {X 0,Y 568.192,Z 280.02,A -85,B 0,C 180,E1 27403.612,E2 27403.612} C_VEL
LIN {X 0,Y 568.183,Z 280.017,A -85,B 0,C 180,E1 27400.225,E2 27400.225} C_VEL
LIN {X 0,Y 568.22,Z 280.018,A -85,B 0,C 180,E1 27396.976,E2 27396.976} C_VEL
LIN {X 0,Y 568.19,Z 280.021,A -85,B 0,C 180,E1 27393.658,E2 27393.658} C_VEL
LIN {X 0,Y 568.188,Z 280.018,A -85,B 0,C 180,E1 27390.227,E2 27390.227} C_VEL
LIN {X 0,Y 568.209,Z 280.198,A -85,B 0,C 180,E1 27387.767,E2 27387.767} C_VEL
LIN {X 0,Y 569.909,Z 287.408,A -85,B 0,C 180,E1 27386.855,E2 27386.855} C_VEL
LIN {X 0,Y 569.505,Z 315.163,A -85,B 0,C 180,E1 27383.704,E2 27383.704} C_VEL
LIN {X 0,Y 569.078,Z 345.224,A -85,B 0,C 180,E1 27380.356,E2 27380.356} C_VEL
LIN {X 0,Y 568.732,Z 376.427,A -85,B 0,C 180,E1 27376.966,E2 27376.966} C_VEL
LIN {X 0,Y 568.504,Z 405.113,A -85,B 0,C 180,E1 27373.93,E2 27373.93} C_VEL
LIN {X 0,Y 568.974,Z 412.425,A -85,B 0,C 180,E1 27373.825,E2 27373.825} C_VEL
LIN {X 0,Y 568.771,Z 516.498,A -85,B 0,C 180,E1 27372.48,E2 27372.48} C_VEL
LIN {X 0,Y 568.682,Z 531.352,A -85,B 0,C 180,E1 27372.101,E2 27372.101} C_VEL
LIN {X 0,Y 568.546,Z 546.158,A -85,B 0,C 180,E1 27371.512,E2 27371.512} C_VEL
LIN {X 0,Y 568.401,Z 559.19,A -85,B 0,C 180,E1 27370.796,E2 27370.796} C_VEL
LIN {X 0,Y 568.285,Z 571.38,A -85,B 0,C 180,E1 27369.927,E2 27369.927} C_VEL
LIN {X 0,Y 568.152,Z 583.55,A -85,B 0,C 180,E1 27368.805,E2 27368.805} C_VEL
LIN {X 0,Y 568.049,Z 593.793,A -85,B 0,C 180,E1 27367.584,E2 27367.584} C_VEL
LIN {X 0,Y 567.983,Z 601.774,A -85,B 0,C 180,E1 27366.366,E2 27366.366} C_VEL
LIN {X 0,Y 567.941,Z 608.857,A -85,B 0,C 180,E1 27364.947,E2 27364.947} C_VEL
LIN {X 0,Y 567.925,Z 614.257,A -85,B 0,C 180,E1 27363.402,E2 27363.402} C_VEL
LIN {X 0,Y 567.916,Z 617.463,A -85,B 0,C 180,E1 27361.915,E2 27361.915} C_VEL
LIN {X 0,Y 567.918,Z 618.907,A -85,B 0,C 180,E1 27360.402,E2 27360.402} C_VEL
LIN {X 0,Y 567.914,Z 618.547,A -85,B 0,C 180,E1 27358.889,E2 27358.889} C_VEL
LIN {X 0,Y 567.918,Z 616.345,A -85,B 0,C 180,E1 27357.375,E2 27357.375} C_VEL
LIN {X 0,Y 567.926,Z 612.593,A -85,B 0,C 180,E1 27355.96,E2 27355.96} C_VEL
LIN {X 0,Y 567.954,Z 606.515,A -85,B 0,C 180,E1 27354.442,E2 27354.442} C_VEL
LIN {X 0,Y 568.002,Z 599.234,A -85,B 0,C 180,E1 27353.124,E2 27353.124} C_VEL
LIN {X 0,Y 568.079,Z 590.545,A -85,B 0,C 180,E1 27351.904,E2 27351.904} C_VEL
LIN {X 0,Y 568.193,Z 579.861,A -85,B 0,C 180,E1 27350.733,E2 27350.733} C_VEL
LIN {X 0,Y 568.306,Z 567.883,A -85,B 0,C 180,E1 27349.712,E2 27349.712} C_VEL
LIN {X 0,Y 568.454,Z 555.563,A -85,B 0,C 180,E1 27348.894,E2 27348.894} C_VEL
LIN {X 0,Y 568.583,Z 542.433,A -85,B 0,C 180,E1 27348.229,E2 27348.229} C_VEL
LIN {X 0,Y 568.702,Z 527.951,A -85,B 0,C 180,E1 27347.706,E2 27347.706} C_VEL
LIN {X 0,Y 568.784,Z 513.277,A -85,B 0,C 180,E1 27347.371,E2 27347.371} C_VEL
LIN {X 0,Y 568.749,Z 406.931,A -85,B 0,C 180,E1 27346.009,E2 27346.009} C_VEL
LIN {X 0,Y 568.474,Z 404.548,A -85,B 0,C 180,E1 27345.952,E2 27345.952} C_VEL
LIN {X 0,Y 568.727,Z 373.331,A -85,B 0,C 180,E1 27342.609,E2 27342.609} C_VEL
LIN {X 0,Y 569.101,Z 343.647,A -85,B 0,C 180,E1 27339.373,E2 27339.373} C_VEL
LIN {X 0,Y 569.599,Z 315.594,A -85,B 0,C 180,E1 27336.187,E2 27336.187} C_VEL
LIN {X 0,Y 570.186,Z 287.767,A -85,B 0,C 180,E1 27332.977,E2 27332.977} C_VEL
LIN {X 0,Y 568.184,Z 280.023,A -85,B 0,C 180,E1 27331.917,E2 27331.917} C_VEL
LIN {X 0,Y 568.221,Z 280.021,A -85,B 0,C 180,E1 27328.728,E2 27328.728} C_VEL
LIN {X 0,Y 568.197,Z 280.021,A -85,B 0,C 180,E1 27325.442,E2 27325.442} C_VEL
LIN {X 0,Y 568.208,Z 280.016,A -85,B 0,C 180,E1 27322.031,E2 27322.031} C_VEL
LIN {X 0,Y 568.202,Z 280.019,A -85,B 0,C 180,E1 27318.842,E2 27318.842} C_VEL
LIN {X 0,Y 568.219,Z 280.022,A -85,B 0,C 180,E1 27315.545,E2 27315.545} C_VEL
LIN {X 0,Y 568.221,Z 280.016,A -85,B 0,C 180,E1 27312.199,E2 27312.199} C_VEL
LIN {X 0,Y 568.174,Z 280.021,A -85,B 0,C 180,E1 27308.921,E2 27308.921} C_VEL
LIN {X 0,Y 568.206,Z 280.023,A -85,B 0,C 180,E1 27305.748,E2 27305.748} C_VEL
LIN {X 0,Y 568.173,Z 280.025,A -85,B 0,C 180,E1 27302.582,E2 27302.582} C_VEL
LIN {X 0,Y 568.184,Z 280.141,A -85,B 0,C 180,E1 27301.617,E2 27301.617} C_VEL
LIN {X 0,Y 571.379,Z 290.409,A -85,B 0,C 180,E1 27300.671,E2 27300.671} C_VEL
LIN {X 0,Y 570.961,Z 331.39,A -85,B 0,C 180,E1 27297.764,E2 27297.764} C_VEL
LIN {X 0,Y 570.326,Z 377.183,A -85,B 0,C 180,E1 27294.551,E2 27294.551} C_VEL
LIN {X 0,Y 570.291,Z 387.17,A -85,B 0,C 180,E1 27293.884,E2 27293.884} C_VEL
LIN {X 0,Y 571.041,Z 394.06,A -85,B 0,C 180,E1 27293.758,E2 27293.758} C_VEL
LIN {X 0,Y 570.358,Z 596.285,A -85,B 0,C 180,E1 27291.062,E2 27291.062} C_VEL
LIN {X 0,Y 570.166,Z 615.325,A -85,B 0,C 180,E1 27290.616,E2 27290.616} C_VEL
LIN {X 0,Y 569.931,Z 633.382,A -85,B 0,C 180,E1 27290.005,E2 27290.005} C_VEL
LIN {X 0,Y 569.648,Z 651.107,A -85,B 0,C 180,E1 27289.211,E2 27289.211} C_VEL
LIN {X 0,Y 569.353,Z 667.763,A -85,B 0,C 180,E1 27288.269,E2 27288.269} C_VEL
LIN {X 0,Y 569.054,Z 683.62,A -85,B 0,C 180,E1 27287.169,E2 27287.169} C_VEL
LIN {X 0,Y 568.769,Z 698.55,A -85,B 0,C 180,E1 27285.917,E2 27285.917} C_VEL
LIN {X 0,Y 568.522,Z 712.013,A -85,B 0,C 180,E1 27284.567,E2 27284.567} C_VEL
LIN {X 0,Y 568.307,Z 724.907,A -85,B 0,C 180,E1 27283.015,E2 27283.015} C_VEL
LIN {X 0,Y 568.149,Z 736.225,A -85,B 0,C 180,E1 27281.368,E2 27281.368} C_VEL
LIN {X 0,Y 568.034,Z 745.991,A -85,B 0,C 180,E1 27279.627,E2 27279.627} C_VEL
LIN {X 0,Y 567.966,Z 753.77,A -85,B 0,C 180,E1 27277.893,E2 27277.893} C_VEL
LIN {X 0,Y 567.931,Z 760.108,A -85,B 0,C 180,E1 27276.064,E2 27276.064} C_VEL
LIN {X 0,Y 567.914,Z 764.875,A -85,B 0,C 180,E1 27274.14,E2 27274.14} C_VEL
LIN {X 0,Y 567.912,Z 767.79,A -85,B 0,C 180,E1 27272.221,E2 27272.221} C_VEL
LIN {X 0,Y 567.908,Z 768.939,A -85,B 0,C 180,E1 27270.303,E2 27270.303} C_VEL
LIN {X 0,Y 567.914,Z 768.416,A -85,B 0,C 180,E1 27268.487,E2 27268.487} C_VEL
LIN {X 0,Y 567.908,Z 766.165,A -85,B 0,C 180,E1 27266.569,E2 27266.569} C_VEL
LIN {X 0,Y 567.926,Z 762.353,A -85,B 0,C 180,E1 27264.748,E2 27264.748} C_VEL
LIN {X 0,Y 567.952,Z 756.823,A -85,B 0,C 180,E1 27262.922,E2 27262.922} C_VEL
LIN {X 0,Y 568,Z 749.43,A -85,B 0,C 180,E1 27261.089,E2 27261.089} C_VEL
LIN {X 0,Y 568.092,Z 740.52,A -85,B 0,C 180,E1 27259.351,E2 27259.351} C_VEL
LIN {X 0,Y 568.23,Z 730.157,A -85,B 0,C 180,E1 27257.708,E2 27257.708} C_VEL
LIN {X 0,Y 568.414,Z 718.357,A -85,B 0,C 180,E1 27256.16,E2 27256.16} C_VEL
LIN {X 0,Y 568.647,Z 705.091,A -85,B 0,C 180,E1 27254.708,E2 27254.708} C_VEL
LIN {X 0,Y 568.927,Z 690.236,A -85,B 0,C 180,E1 27253.355,E2 27253.355} C_VEL
LIN {X 0,Y 569.234,Z 674.322,A -85,B 0,C 180,E1 27252.157,E2 27252.157} C_VEL
LIN {X 0,Y 569.54,Z 657.161,A -85,B 0,C 180,E1 27251.107,E2 27251.107} C_VEL
LIN {X 0,Y 569.833,Z 639.824,A -85,B 0,C 180,E1 27250.26,E2 27250.26} C_VEL
LIN {X 0,Y 570.098,Z 621.554,A -85,B 0,C 180,E1 27249.574,E2 27249.574} C_VEL
LIN {X 0,Y 570.297,Z 603.079,A -85,B 0,C 180,E1 27249.076,E2 27249.076} C_VEL
LIN {X 0,Y 570.426,Z 582.939,A -85,B 0,C 180,E1 27248.737,E2 27248.737} C_VEL
LIN {X 0,Y 570.88,Z 390.97,A -85,B 0,C 180,E1 27246.193,E2 27246.193} C_VEL
LIN {X 0,Y 570.222,Z 386.265,A -85,B 0,C 180,E1 27246.079,E2 27246.079} C_VEL
LIN {X 0,Y 570.892,Z 338.613,A -85,B 0,C 180,E1 27242.744,E2 27242.744} C_VEL
LIN {X 0,Y 571.389,Z 295.613,A -85,B 0,C 180,E1 27239.68,E2 27239.68} C_VEL
LIN {X 0,Y 571.361,Z 289.472,A -85,B 0,C 180,E1 27239.231,E2 27239.231} C_VEL
LIN {X 0,Y 568.157,Z 280.027,A -85,B 0,C 180,E1 27238.342,E2 27238.342} C_VEL
LIN {X 0,Y 568.145,Z 280.024,A -85,B 0,C 180,E1 27235.095,E2 27235.095} C_VEL
LIN {X 0,Y 568.191,Z 280.024,A -85,B 0,C 180,E1 27231.984,E2 27231.984} C_VEL
LIN {X 0,Y 568.135,Z 280.023,A -85,B 0,C 180,E1 27228.838,E2 27228.838} C_VEL
LIN {X 0,Y 568.205,Z 280.023,A -85,B 0,C 180,E1 27225.687,E2 27225.687} C_VEL
LIN {X 0,Y 568.135,Z 280.022,A -85,B 0,C 180,E1 27222.64,E2 27222.64} C_VEL
LIN {X 0,Y 568.177,Z 280.022,A -85,B 0,C 180,E1 27219.419,E2 27219.419} C_VEL
LIN {X 0,Y 568.14,Z 280.022,A -85,B 0,C 180,E1 27216.462,E2 27216.462} C_VEL
LIN {X 0,Y 568.151,Z 280.022,A -85,B 0,C 180,E1 27213.105,E2 27213.105} C_VEL
LIN {X 0,Y 568.169,Z 280.022,A -85,B 0,C 180,E1 27210.103,E2 27210.103} C_VEL
LIN {X 0,Y 568.14,Z 280.022,A -85,B 0,C 180,E1 27206.844,E2 27206.844} C_VEL
LIN {X 0,Y 568.209,Z 280.022,A -85,B 0,C 180,E1 27203.765,E2 27203.765} C_VEL
LIN {X 0,Y 568.142,Z 280.021,A -85,B 0,C 180,E1 27200.571,E2 27200.571} C_VEL
LIN {X 0,Y 568.193,Z 280.021,A -85,B 0,C 180,E1 27197.408,E2 27197.408} C_VEL
LIN {X 0,Y 568.149,Z 280.021,A -85,B 0,C 180,E1 27194.369,E2 27194.369} C_VEL
LIN {X 0,Y 568.153,Z 280.021,A -85,B 0,C 180,E1 27190.958,E2 27190.958} C_VEL
LIN {X 0,Y 568.188,Z 280.022,A -85,B 0,C 180,E1 27187.891,E2 27187.891} C_VEL
LIN {X 0,Y 568.147,Z 280.021,A -85,B 0,C 180,E1 27184.746,E2 27184.746} C_VEL
LIN {X 0,Y 568.216,Z 280.022,A -85,B 0,C 180,E1 27181.615,E2 27181.615} C_VEL
LIN {X 0,Y 568.147,Z 280.021,A -85,B 0,C 180,E1 27178.489,E2 27178.489} C_VEL
LIN {X 0,Y 568.191,Z 280.019,A -85,B 0,C 180,E1 27175.257,E2 27175.257} C_VEL
LIN {X 0,Y 568.158,Z 280.021,A -85,B 0,C 180,E1 27172.206,E2 27172.206} C_VEL
LIN {X 0,Y 568.158,Z 280.02,A -85,B 0,C 180,E1 27168.84,E2 27168.84} C_VEL
LIN {X 0,Y 568.2,Z 280.022,A -85,B 0,C 180,E1 27165.74,E2 27165.74} C_VEL
LIN {X 0,Y 568.151,Z 280.02,A -85,B 0,C 180,E1 27162.519,E2 27162.519} C_VEL
LIN {X 0,Y 568.182,Z 280.021,A -85,B 0,C 180,E1 27159.894,E2 27159.894} C_VEL
LIN {X 0,Y 567.239,Z 280.145,A -85,B 0,C 180,E1 27159.117,E2 27159.117} C_VEL
LIN {X 0,Y 560.749,Z 280.945,A -85,B 0,C 180,E1 27156.936,E2 27156.936} C_VEL
LIN {X 0,Y 560.214,Z 281.009,A -85,B 0,C 180,E1 27156.368,E2 27156.368} C_VEL
LIN {X 0,Y 560.258,Z 281.007,A -85,B 0,C 180,E1 27153.161,E2 27153.161} C_VEL
LIN {X 0,Y 560.231,Z 281.01,A -85,B 0,C 180,E1 27150.021,E2 27150.021} C_VEL
LIN {X 0,Y 560.22,Z 281.008,A -85,B 0,C 180,E1 27146.642,E2 27146.642} C_VEL
LIN {X 0,Y 560.282,Z 281.008,A -85,B 0,C 180,E1 27143.416,E2 27143.416} C_VEL
LIN {X 0,Y 560.219,Z 281.009,A -85,B 0,C 180,E1 27140.283,E2 27140.283} C_VEL
LIN {X 0,Y 560.254,Z 281.006,A -85,B 0,C 180,E1 27137.024,E2 27137.024} C_VEL
LIN {X 0,Y 560.242,Z 281.01,A -85,B 0,C 180,E1 27133.865,E2 27133.865} C_VEL
LIN {X 0,Y 560.227,Z 281.007,A -85,B 0,C 180,E1 27130.648,E2 27130.648} C_VEL
LIN {X 0,Y 560.277,Z 281.011,A -85,B 0,C 180,E1 27127.483,E2 27127.483} C_VEL
LIN {X 0,Y 560.224,Z 281.008,A -85,B 0,C 180,E1 27124.207,E2 27124.207} C_VEL
LIN {X 0,Y 560.253,Z 281.006,A -85,B 0,C 180,E1 27120.928,E2 27120.928} C_VEL
LIN {X 0,Y 560.253,Z 281.01,A -85,B 0,C 180,E1 27117.731,E2 27117.731} C_VEL
LIN {X 0,Y 560.226,Z 281.007,A -85,B 0,C 180,E1 27114.459,E2 27114.459} C_VEL
LIN {X 0,Y 560.285,Z 281.006,A -85,B 0,C 180,E1 27111.238,E2 27111.238} C_VEL
LIN {X 0,Y 560.233,Z 281.009,A -85,B 0,C 180,E1 27107.972,E2 27107.972} C_VEL
LIN {X 0,Y 560.235,Z 281.006,A -85,B 0,C 180,E1 27104.574,E2 27104.574} C_VEL
LIN {X 0,Y 560.284,Z 281.008,A -85,B 0,C 180,E1 27101.32,E2 27101.32} C_VEL
LIN {X 0,Y 560.228,Z 281.008,A -85,B 0,C 180,E1 27098.105,E2 27098.105} C_VEL
LIN {X 0,Y 560.256,Z 281.005,A -85,B 0,C 180,E1 27094.811,E2 27094.811} C_VEL
LIN {X 0,Y 560.257,Z 281.01,A -85,B 0,C 180,E1 27091.635,E2 27091.635} C_VEL
LIN {X 0,Y 560.232,Z 281.007,A -85,B 0,C 180,E1 27088.363,E2 27088.363} C_VEL
LIN {X 0,Y 560.283,Z 281.005,A -85,B 0,C 180,E1 27085.085,E2 27085.085} C_VEL
LIN {X 0,Y 560.237,Z 281.008,A -85,B 0,C 180,E1 27081.894,E2 27081.894} C_VEL
LIN {X 0,Y 560.239,Z 281.006,A -85,B 0,C 180,E1 27078.451,E2 27078.451} C_VEL
LIN {X 0,Y 560.285,Z 281.007,A -85,B 0,C 180,E1 27075.214,E2 27075.214} C_VEL
LIN {X 0,Y 560.236,Z 281.007,A -85,B 0,C 180,E1 27072.015,E2 27072.015} C_VEL
LIN {X 0,Y 560.261,Z 281.004,A -85,B 0,C 180,E1 27068.675,E2 27068.675} C_VEL
LIN {X 0,Y 560.271,Z 281.011,A -85,B 0,C 180,E1 27065.429,E2 27065.429} C_VEL
LIN {X 0,Y 560.236,Z 281.006,A -85,B 0,C 180,E1 27062.121,E2 27062.121} C_VEL
LIN {X 0,Y 560.281,Z 281.003,A -85,B 0,C 180,E1 27058.833,E2 27058.833} C_VEL
LIN {X 0,Y 560.262,Z 281.009,A -85,B 0,C 180,E1 27055.533,E2 27055.533} C_VEL
LIN {X 0,Y 560.241,Z 281.005,A -85,B 0,C 180,E1 27052.239,E2 27052.239} C_VEL
LIN {X 0,Y 560.282,Z 281.006,A -85,B 0,C 180,E1 27049.01,E2 27049.01} C_VEL
LIN {X 0,Y 560.249,Z 281.008,A -85,B 0,C 180,E1 27045.693,E2 27045.693} C_VEL
LIN {X 0,Y 560.247,Z 281.005,A -85,B 0,C 180,E1 27042.282,E2 27042.282} C_VEL
LIN {X 0,Y 560.283,Z 281.008,A -85,B 0,C 180,E1 27039.043,E2 27039.043} C_VEL
LIN {X 0,Y 560.248,Z 281.009,A -85,B 0,C 180,E1 27035.701,E2 27035.701} C_VEL
LIN {X 0,Y 560.247,Z 281.005,A -85,B 0,C 180,E1 27032.248,E2 27032.248} C_VEL
LIN {X 0,Y 560.282,Z 281.012,A -85,B 0,C 180,E1 27029.021,E2 27029.021} C_VEL
LIN {X 0,Y 560.269,Z 281.186,A -85,B 0,C 180,E1 27028.081,E2 27028.081} C_VEL
LIN {X 0,Y 562.32,Z 289.896,A -85,B 0,C 180,E1 27026.961,E2 27026.961} C_VEL
LIN {X 0,Y 561.848,Z 317.139,A -85,B 0,C 180,E1 27023.834,E2 27023.834} C_VEL
LIN {X 0,Y 561.325,Z 347.28,A -85,B 0,C 180,E1 27020.432,E2 27020.432} C_VEL
LIN {X 0,Y 560.898,Z 377.896,A -85,B 0,C 180,E1 27017.05,E2 27017.05} C_VEL
LIN {X 0,Y 560.633,Z 405.084,A -85,B 0,C 180,E1 27014.131,E2 27014.131} C_VEL
LIN {X 0,Y 561.208,Z 412.603,A -85,B 0,C 180,E1 27014.019,E2 27014.019} C_VEL
LIN {X 0,Y 560.959,Z 516.413,A -85,B 0,C 180,E1 27012.659,E2 27012.659} C_VEL
LIN {X 0,Y 560.852,Z 531.296,A -85,B 0,C 180,E1 27012.275,E2 27012.275} C_VEL
LIN {X 0,Y 560.687,Z 546.174,A -85,B 0,C 180,E1 27011.676,E2 27011.676} C_VEL
LIN {X 0,Y 560.516,Z 559.199,A -85,B 0,C 180,E1 27010.95,E2 27010.95} C_VEL
LIN {X 0,Y 560.366,Z 571.387,A -85,B 0,C 180,E1 27010.069,E2 27010.069} C_VEL
LIN {X 0,Y 560.204,Z 583.557,A -85,B 0,C 180,E1 27008.931,E2 27008.931} C_VEL
LIN {X 0,Y 560.079,Z 593.797,A -85,B 0,C 180,E1 27007.693,E2 27007.693} C_VEL
LIN {X 0,Y 559.999,Z 601.778,A -85,B 0,C 180,E1 27006.457,E2 27006.457} C_VEL
LIN {X 0,Y 559.947,Z 608.859,A -85,B 0,C 180,E1 27005.018,E2 27005.018} C_VEL
LIN {X 0,Y 559.927,Z 614.326,A -85,B 0,C 180,E1 27003.428,E2 27003.428} C_VEL
LIN {X 0,Y 559.916,Z 617.464,A -85,B 0,C 180,E1 27001.943,E2 27001.943} C_VEL
LIN {X 0,Y 559.918,Z 618.907,A -85,B 0,C 180,E1 27000.408,E2 27000.408} C_VEL
LIN {X 0,Y 559.914,Z 618.546,A -85,B 0,C 180,E1 26998.873,E2 26998.873} C_VEL
LIN {X 0,Y 559.918,Z 616.343,A -85,B 0,C 180,E1 26997.337,E2 26997.337} C_VEL
LIN {X 0,Y 559.929,Z 612.591,A -85,B 0,C 180,E1 26995.903,E2 26995.903} C_VEL
LIN {X 0,Y 559.963,Z 606.512,A -85,B 0,C 180,E1 26994.363,E2 26994.363} C_VEL
LIN {X 0,Y 560.023,Z 599.23,A -85,B 0,C 180,E1 26993.025,E2 26993.025} C_VEL
LIN {X 0,Y 560.117,Z 590.54,A -85,B 0,C 180,E1 26991.788,E2 26991.788} C_VEL
LIN {X 0,Y 560.253,Z 579.854,A -85,B 0,C 180,E1 26990.6,E2 26990.6} C_VEL
LIN {X 0,Y 560.396,Z 567.873,A -85,B 0,C 180,E1 26989.565,E2 26989.565} C_VEL
LIN {X 0,Y 560.577,Z 555.554,A -85,B 0,C 180,E1 26988.736,E2 26988.736} C_VEL
LIN {X 0,Y 560.733,Z 542.417,A -85,B 0,C 180,E1 26988.061,E2 26988.061} C_VEL
LIN {X 0,Y 560.876,Z 527.929,A -85,B 0,C 180,E1 26987.532,E2 26987.532} C_VEL
LIN {X 0,Y 560.974,Z 513.234,A -85,B 0,C 180,E1 26987.193,E2 26987.193} C_VEL
LIN {X 0,Y 560.985,Z 407.702,A -85,B 0,C 180,E1 26985.822,E2 26985.822} C_VEL
LIN {X 0,Y 560.595,Z 404.542,A -85,B 0,C 180,E1 26985.75,E2 26985.75} C_VEL
LIN {X 0,Y 560.912,Z 373.812,A -85,B 0,C 180,E1 26982.412,E2 26982.412} C_VEL
LIN {X 0,Y 561.491,Z 344.349,A -85,B 0,C 180,E1 26979.081,E2 26979.081} C_VEL
LIN {X 0,Y 562.114,Z 316.27,A -85,B 0,C 180,E1 26975.85,E2 26975.85} C_VEL
LIN {X 0,Y 562.694,Z 290.036,A -85,B 0,C 180,E1 26972.795,E2 26972.795} C_VEL
LIN {X 0,Y 560.237,Z 281.014,A -85,B 0,C 180,E1 26971.541,E2 26971.541} C_VEL
LIN {X 0,Y 560.277,Z 281.006,A -85,B 0,C 180,E1 26968.233,E2 26968.233} C_VEL
LIN {X 0,Y 560.279,Z 281.01,A -85,B 0,C 180,E1 26964.925,E2 26964.925} C_VEL
LIN {X 0,Y 560.266,Z 281.01,A -85,B 0,C 180,E1 26961.578,E2 26961.578} C_VEL
LIN {X 0,Y 560.281,Z 281.004,A -85,B 0,C 180,E1 26958.241,E2 26958.241} C_VEL
LIN {X 0,Y 560.254,Z 281.009,A -85,B 0,C 180,E1 26954.886,E2 26954.886} C_VEL
LIN {X 0,Y 560.28,Z 281.011,A -85,B 0,C 180,E1 26951.596,E2 26951.596} C_VEL
LIN {X 0,Y 560.276,Z 281.007,A -85,B 0,C 180,E1 26948.259,E2 26948.259} C_VEL
LIN {X 0,Y 560.224,Z 281.013,A -85,B 0,C 180,E1 26944.995,E2 26944.995} C_VEL
LIN {X 0,Y 560.28,Z 281.051,A -85,B 0,C 180,E1 26942.024,E2 26942.024} C_VEL
LIN {X 0,Y 564.035,Z 292.97,A -85,B 0,C 180,E1 26940.883,E2 26940.883} C_VEL
LIN {X 0,Y 563.444,Z 332.903,A -85,B 0,C 180,E1 26937.994,E2 26937.994} C_VEL
LIN {X 0,Y 562.894,Z 375.608,A -85,B 0,C 180,E1 26935.009,E2 26935.009} C_VEL
LIN {X 0,Y 562.802,Z 387.139,A -85,B 0,C 180,E1 26934.223,E2 26934.223} C_VEL
LIN {X 0,Y 563.716,Z 395.074,A -85,B 0,C 180,E1 26934.072,E2 26934.072} C_VEL
LIN {X 0,Y 562.891,Z 596.285,A -85,B 0,C 180,E1 26931.355,E2 26931.355} C_VEL
LIN {X 0,Y 562.66,Z 615.31,A -85,B 0,C 180,E1 26930.904,E2 26930.904} C_VEL
LIN {X 0,Y 562.376,Z 633.38,A -85,B 0,C 180,E1 26930.286,E2 26930.286} C_VEL
LIN {X 0,Y 562.03,Z 651.129,A -85,B 0,C 180,E1 26929.481,E2 26929.481} C_VEL
LIN {X 0,Y 561.671,Z 667.76,A -85,B 0,C 180,E1 26928.528,E2 26928.528} C_VEL
LIN {X 0,Y 561.31,Z 683.617,A -85,B 0,C 180,E1 26927.414,E2 26927.414} C_VEL
LIN {X 0,Y 560.962,Z 698.549,A -85,B 0,C 180,E1 26926.145,E2 26926.145} C_VEL
LIN {X 0,Y 560.663,Z 712.012,A -85,B 0,C 180,E1 26924.775,E2 26924.775} C_VEL
LIN {X 0,Y 560.401,Z 724.908,A -85,B 0,C 180,E1 26923.202,E2 26923.202} C_VEL
LIN {X 0,Y 560.204,Z 736.315,A -85,B 0,C 180,E1 26921.517,E2 26921.517} C_VEL
LIN {X 0,Y 560.067,Z 745.99,A -85,B 0,C 180,E1 26919.765,E2 26919.765} C_VEL
LIN {X 0,Y 559.98,Z 753.769,A -85,B 0,C 180,E1 26918.006,E2 26918.006} C_VEL
LIN {X 0,Y 559.936,Z 760.108,A -85,B 0,C 180,E1 26916.151,E2 26916.151} C_VEL
LIN {X 0,Y 559.914,Z 764.876,A -85,B 0,C 180,E1 26914.199,E2 26914.199} C_VEL
LIN {X 0,Y 559.912,Z 767.791,A -85,B 0,C 180,E1 26912.252,E2 26912.252} C_VEL
LIN {X 0,Y 559.908,Z 768.939,A -85,B 0,C 180,E1 26910.308,E2 26910.308} C_VEL
LIN {X 0,Y 559.913,Z 768.416,A -85,B 0,C 180,E1 26908.466,E2 26908.466} C_VEL
LIN {X 0,Y 559.909,Z 766.164,A -85,B 0,C 180,E1 26906.52,E2 26906.52} C_VEL
LIN {X 0,Y 559.928,Z 762.353,A -85,B 0,C 180,E1 26904.673,E2 26904.673} C_VEL
LIN {X 0,Y 559.961,Z 756.823,A -85,B 0,C 180,E1 26902.821,E2 26902.821} C_VEL
LIN {X 0,Y 560.027,Z 749.431,A -85,B 0,C 180,E1 26900.961,E2 26900.961} C_VEL
LIN {X 0,Y 560.136,Z 740.521,A -85,B 0,C 180,E1 26899.198,E2 26899.198} C_VEL
LIN {X 0,Y 560.307,Z 730.158,A -85,B 0,C 180,E1 26897.531,E2 26897.531} C_VEL
LIN {X 0,Y 560.531,Z 718.358,A -85,B 0,C 180,E1 26895.961,E2 26895.961} C_VEL
LIN {X 0,Y 560.822,Z 704.809,A -85,B 0,C 180,E1 26894.46,E2 26894.46} C_VEL
LIN {X 0,Y 561.16,Z 690.039,A -85,B 0,C 180,E1 26893.1,E2 26893.1} C_VEL
LIN {X 0,Y 561.529,Z 674.245,A -85,B 0,C 180,E1 26891.899,E2 26891.899} C_VEL
LIN {X 0,Y 561.9,Z 657.064,A -85,B 0,C 180,E1 26890.835,E2 26890.835} C_VEL
LIN {X 0,Y 562.254,Z 639.826,A -85,B 0,C 180,E1 26889.982,E2 26889.982} C_VEL
LIN {X 0,Y 562.571,Z 621.558,A -85,B 0,C 180,E1 26889.288,E2 26889.288} C_VEL
LIN {X 0,Y 562.815,Z 603.04,A -85,B 0,C 180,E1 26888.784,E2 26888.784} C_VEL
LIN {X 0,Y 562.972,Z 582.811,A -85,B 0,C 180,E1 26888.439,E2 26888.439} C_VEL
LIN {X 0,Y 563.553,Z 391.996,A -85,B 0,C 180,E1 26885.878,E2 26885.878} C_VEL
LIN {X 0,Y 562.736,Z 386.265,A -85,B 0,C 180,E1 26885.741,E2 26885.741} C_VEL
LIN {X 0,Y 563.503,Z 338.272,A -85,B 0,C 180,E1 26882.35,E2 26882.35} C_VEL
LIN {X 0,Y 564.121,Z 296.118,A -85,B 0,C 180,E1 26879.307,E2 26879.307} C_VEL
LIN {X 0,Y 563.993,Z 292.073,A -85,B 0,C 180,E1 26879,E2 26879} C_VEL
LIN {X 0,Y 560.263,Z 281.013,A -85,B 0,C 180,E1 26877.933,E2 26877.933} C_VEL
LIN {X 0,Y 560.199,Z 281.014,A -85,B 0,C 180,E1 26874.796,E2 26874.796} C_VEL
LIN {X 0,Y 560.253,Z 281.012,A -85,B 0,C 180,E1 26871.579,E2 26871.579} C_VEL
LIN {X 0,Y 560.201,Z 281.013,A -85,B 0,C 180,E1 26868.536,E2 26868.536} C_VEL
LIN {X 0,Y 560.212,Z 281.012,A -85,B 0,C 180,E1 26865.173,E2 26865.173} C_VEL
LIN {X 0,Y 560.227,Z 281.011,A -85,B 0,C 180,E1 26862.15,E2 26862.15} C_VEL
LIN {X 0,Y 560.2,Z 281.011,A -85,B 0,C 180,E1 26858.907,E2 26858.907} C_VEL
LIN {X 0,Y 560.272,Z 281.012,A -85,B 0,C 180,E1 26855.711,E2 26855.711} C_VEL
LIN {X 0,Y 560.202,Z 281.011,A -85,B 0,C 180,E1 26852.496,E2 26852.496} C_VEL
LIN {X 0,Y 560.221,Z 281.01,A -85,B 0,C 180,E1 26849.16,E2 26849.16} C_VEL
LIN {X 0,Y 560.225,Z 281.011,A -85,B 0,C 180,E1 26846.142,E2 26846.142} C_VEL
LIN {X 0,Y 560.207,Z 281.01,A -85,B 0,C 180,E1 26842.899,E2 26842.899} C_VEL
LIN {X 0,Y 560.271,Z 281.012,A -85,B 0,C 180,E1 26839.713,E2 26839.713} C_VEL
LIN {X 0,Y 560.204,Z 281.01,A -85,B 0,C 180,E1 26836.579,E2 26836.579} C_VEL
LIN {X 0,Y 560.257,Z 281.009,A -85,B 0,C 180,E1 26833.416,E2 26833.416} C_VEL
LIN {X 0,Y 560.214,Z 281.01,A -85,B 0,C 180,E1 26830.282,E2 26830.282} C_VEL
LIN {X 0,Y 560.213,Z 281.009,A -85,B 0,C 180,E1 26826.869,E2 26826.869} C_VEL
LIN {X 0,Y 560.271,Z 281.011,A -85,B 0,C 180,E1 26823.685,E2 26823.685} C_VEL
LIN {X 0,Y 560.207,Z 281.01,A -85,B 0,C 180,E1 26820.513,E2 26820.513} C_VEL
LIN {X 0,Y 560.26,Z 281.008,A -85,B 0,C 180,E1 26817.342,E2 26817.342} C_VEL
LIN {X 0,Y 560.221,Z 281.01,A -85,B 0,C 180,E1 26814.163,E2 26814.163} C_VEL
LIN {X 0,Y 560.22,Z 281.009,A -85,B 0,C 180,E1 26810.862,E2 26810.862} C_VEL
LIN {X 0,Y 560.262,Z 281.011,A -85,B 0,C 180,E1 26807.74,E2 26807.74} C_VEL
LIN {X 0,Y 560.212,Z 281.009,A -85,B 0,C 180,E1 26804.529,E2 26804.529} C_VEL
LIN {X 0,Y 560.274,Z 281.008,A -85,B 0,C 180,E1 26801.369,E2 26801.369} C_VEL
LIN {X 0,Y 560.219,Z 281.01,A -85,B 0,C 180,E1 26798.211,E2 26798.211} C_VEL
LIN {X 0,Y 560.214,Z 281.009,A -85,B 0,C 180,E1 26796.368,E2 26796.368} C_VEL
LIN {X 0,Y 559.244,Z 281.14,A -85,B 0,C 180,E1 26795.58,E2 26795.58} C_VEL
LIN {X 0,Y 552.743,Z 281.945,A -85,B 0,C 180,E1 26793.311,E2 26793.311} C_VEL
LIN {X 0,Y 552.286,Z 281.997,A -85,B 0,C 180,E1 26792.792,E2 26792.792} C_VEL
LIN {X 0,Y 552.343,Z 282,A -85,B 0,C 180,E1 26789.548,E2 26789.548} C_VEL
LIN {X 0,Y 552.278,Z 281.998,A -85,B 0,C 180,E1 26786.361,E2 26786.361} C_VEL
LIN {X 0,Y 552.313,Z 281.996,A -85,B 0,C 180,E1 26783.06,E2 26783.06} C_VEL
LIN {X 0,Y 552.297,Z 281.998,A -85,B 0,C 180,E1 26779.975,E2 26779.975} C_VEL
LIN {X 0,Y 552.286,Z 281.997,A -85,B 0,C 180,E1 26776.678,E2 26776.678} C_VEL
LIN {X 0,Y 552.341,Z 281.999,A -85,B 0,C 180,E1 26773.46,E2 26773.46} C_VEL
LIN {X 0,Y 552.285,Z 281.998,A -85,B 0,C 180,E1 26770.187,E2 26770.187} C_VEL
LIN {X 0,Y 552.301,Z 281.996,A -85,B 0,C 180,E1 26766.813,E2 26766.813} C_VEL
LIN {X 0,Y 552.325,Z 281.999,A -85,B 0,C 180,E1 26763.625,E2 26763.625} C_VEL
LIN {X 0,Y 552.284,Z 281.997,A -85,B 0,C 180,E1 26760.337,E2 26760.337} C_VEL
LIN {X 0,Y 552.33,Z 281.994,A -85,B 0,C 180,E1 26757.051,E2 26757.051} C_VEL
LIN {X 0,Y 552.306,Z 281.998,A -85,B 0,C 180,E1 26753.809,E2 26753.809} C_VEL
LIN {X 0,Y 552.289,Z 281.996,A -85,B 0,C 180,E1 26750.45,E2 26750.45} C_VEL
LIN {X 0,Y 552.341,Z 281.995,A -85,B 0,C 180,E1 26747.161,E2 26747.161} C_VEL
LIN {X 0,Y 552.298,Z 281.998,A -85,B 0,C 180,E1 26743.932,E2 26743.932} C_VEL
LIN {X 0,Y 552.296,Z 281.995,A -85,B 0,C 180,E1 26740.535,E2 26740.535} C_VEL
LIN {X 0,Y 552.347,Z 281.996,A -85,B 0,C 180,E1 26737.279,E2 26737.279} C_VEL
LIN {X 0,Y 552.292,Z 281.997,A -85,B 0,C 180,E1 26734.048,E2 26734.048} C_VEL
LIN {X 0,Y 552.314,Z 281.994,A -85,B 0,C 180,E1 26730.725,E2 26730.725} C_VEL
LIN {X 0,Y 552.33,Z 281.999,A -85,B 0,C 180,E1 26727.509,E2 26727.509} C_VEL
LIN {X 0,Y 552.292,Z 281.996,A -85,B 0,C 180,E1 26724.181,E2 26724.181} C_VEL
LIN {X 0,Y 552.34,Z 281.993,A -85,B 0,C 180,E1 26720.938,E2 26720.938} C_VEL
LIN {X 0,Y 552.314,Z 281.998,A -85,B 0,C 180,E1 26717.665,E2 26717.665} C_VEL
LIN {X 0,Y 552.298,Z 281.995,A -85,B 0,C 180,E1 26714.35,E2 26714.35} C_VEL
LIN {X 0,Y 552.345,Z 281.995,A -85,B 0,C 180,E1 26711.093,E2 26711.093} C_VEL
LIN {X 0,Y 552.301,Z 281.997,A -85,B 0,C 180,E1 26707.879,E2 26707.879} C_VEL
LIN {X 0,Y 552.309,Z 281.994,A -85,B 0,C 180,E1 26704.477,E2 26704.477} C_VEL
LIN {X 0,Y 552.345,Z 281.996,A -85,B 0,C 180,E1 26701.175,E2 26701.175} C_VEL
LIN {X 0,Y 552.301,Z 281.996,A -85,B 0,C 180,E1 26697.908,E2 26697.908} C_VEL
LIN {X 0,Y 552.318,Z 281.993,A -85,B 0,C 180,E1 26694.547,E2 26694.547} C_VEL
LIN {X 0,Y 552.345,Z 281.998,A -85,B 0,C 180,E1 26691.219,E2 26691.219} C_VEL
LIN {X 0,Y 552.301,Z 281.996,A -85,B 0,C 180,E1 26687.919,E2 26687.919} C_VEL
LIN {X 0,Y 552.331,Z 281.992,A -85,B 0,C 180,E1 26684.615,E2 26684.615} C_VEL
LIN {X 0,Y 552.343,Z 281.999,A -85,B 0,C 180,E1 26681.214,E2 26681.214} C_VEL
LIN {X 0,Y 552.303,Z 281.997,A -85,B 0,C 180,E1 26677.878,E2 26677.878} C_VEL
LIN {X 0,Y 552.328,Z 281.994,A -85,B 0,C 180,E1 26674.512,E2 26674.512} C_VEL
LIN {X 0,Y 552.344,Z 281.998,A -85,B 0,C 180,E1 26671.177,E2 26671.177} C_VEL
LIN {X 0,Y 552.338,Z 282.112,A -85,B 0,C 180,E1 26668.412,E2 26668.412} C_VEL
LIN {X 0,Y 554.732,Z 292.33,A -85,B 0,C 180,E1 26667.076,E2 26667.076} C_VEL
LIN {X 0,Y 554.2,Z 318.806,A -85,B 0,C 180,E1 26664.004,E2 26664.004} C_VEL
LIN {X 0,Y 553.586,Z 348.859,A -85,B 0,C 180,E1 26660.565,E2 26660.565} C_VEL
LIN {X 0,Y 553.074,Z 379.428,A -85,B 0,C 180,E1 26657.136,E2 26657.136} C_VEL
LIN {X 0,Y 552.756,Z 405.029,A -85,B 0,C 180,E1 26654.338,E2 26654.338} C_VEL
LIN {X 0,Y 553.447,Z 412.909,A -85,B 0,C 180,E1 26654.216,E2 26654.216} C_VEL
LIN {X 0,Y 553.152,Z 516.461,A -85,B 0,C 180,E1 26652.841,E2 26652.841} C_VEL
LIN {X 0,Y 553.026,Z 531.39,A -85,B 0,C 180,E1 26652.449,E2 26652.449} C_VEL
LIN {X 0,Y 552.834,Z 546.189,A -85,B 0,C 180,E1 26651.844,E2 26651.844} C_VEL
LIN {X 0,Y 552.638,Z 559.012,A -85,B 0,C 180,E1 26651.12,E2 26651.12} C_VEL
LIN {X 0,Y 552.451,Z 571.394,A -85,B 0,C 180,E1 26650.215,E2 26650.215} C_VEL
LIN {X 0,Y 552.261,Z 583.563,A -85,B 0,C 180,E1 26649.061,E2 26649.061} C_VEL
LIN {X 0,Y 552.112,Z 593.801,A -85,B 0,C 180,E1 26647.805,E2 26647.805} C_VEL
LIN {X 0,Y 552.016,Z 601.782,A -85,B 0,C 180,E1 26646.551,E2 26646.551} C_VEL
LIN {X 0,Y 551.953,Z 608.862,A -85,B 0,C 180,E1 26645.091,E2 26645.091} C_VEL
LIN {X 0,Y 551.927,Z 614.179,A -85,B 0,C 180,E1 26643.53,E2 26643.53} C_VEL
LIN {X 0,Y 551.917,Z 617.464,A -85,B 0,C 180,E1 26641.971,E2 26641.971} C_VEL
LIN {X 0,Y 551.918,Z 618.907,A -85,B 0,C 180,E1 26640.414,E2 26640.414} C_VEL
LIN {X 0,Y 551.914,Z 618.545,A -85,B 0,C 180,E1 26638.857,E2 26638.857} C_VEL
LIN {X 0,Y 551.918,Z 616.341,A -85,B 0,C 180,E1 26637.299,E2 26637.299} C_VEL
LIN {X 0,Y 551.932,Z 612.589,A -85,B 0,C 180,E1 26635.843,E2 26635.843} C_VEL
LIN {X 0,Y 551.973,Z 606.509,A -85,B 0,C 180,E1 26634.281,E2 26634.281} C_VEL
LIN {X 0,Y 552.045,Z 599.225,A -85,B 0,C 180,E1 26632.924,E2 26632.924} C_VEL
LIN {X 0,Y 552.157,Z 590.534,A -85,B 0,C 180,E1 26631.669,E2 26631.669} C_VEL
LIN {X 0,Y 552.319,Z 579.847,A -85,B 0,C 180,E1 26630.464,E2 26630.464} C_VEL
LIN {X 0,Y 552.491,Z 567.863,A -85,B 0,C 180,E1 26629.414,E2 26629.414} C_VEL
LIN {X 0,Y 552.705,Z 555.541,A -85,B 0,C 180,E1 26628.574,E2 26628.574} C_VEL
LIN {X 0,Y 552.888,Z 542.401,A -85,B 0,C 180,E1 26627.889,E2 26627.889} C_VEL
LIN {X 0,Y 553.057,Z 527.907,A -85,B 0,C 180,E1 26627.353,E2 26627.353} C_VEL
LIN {X 0,Y 553.172,Z 513.19,A -85,B 0,C 180,E1 26627.009,E2 26627.009} C_VEL
LIN {X 0,Y 553.236,Z 408.546,A -85,B 0,C 180,E1 26625.631,E2 26625.631} C_VEL
LIN {X 0,Y 552.721,Z 404.536,A -85,B 0,C 180,E1 26625.543,E2 26625.543} C_VEL
LIN {X 0,Y 553.21,Z 374.939,A -85,B 0,C 180,E1 26622.214,E2 26622.214} C_VEL
LIN {X 0,Y 553.884,Z 345.505,A -85,B 0,C 180,E1 26618.835,E2 26618.835} C_VEL
LIN {X 0,Y 554.58,Z 317.766,A -85,B 0,C 180,E1 26615.614,E2 26615.614} C_VEL
LIN {X 0,Y 555.289,Z 292.894,A -85,B 0,C 180,E1 26612.666,E2 26612.666} C_VEL
LIN {X 0,Y 552.319,Z 282.002,A -85,B 0,C 180,E1 26611.095,E2 26611.095} C_VEL
LIN {X 0,Y 552.31,Z 281.999,A -85,B 0,C 180,E1 26607.718,E2 26607.718} C_VEL
LIN {X 0,Y 552.341,Z 281.994,A -85,B 0,C 180,E1 26604.345,E2 26604.345} C_VEL
LIN {X 0,Y 552.333,Z 281.999,A -85,B 0,C 180,E1 26600.951,E2 26600.951} C_VEL
LIN {X 0,Y 552.338,Z 281.999,A -85,B 0,C 180,E1 26597.611,E2 26597.611} C_VEL
LIN {X 0,Y 552.342,Z 281.994,A -85,B 0,C 180,E1 26594.182,E2 26594.182} C_VEL
LIN {X 0,Y 552.304,Z 281.999,A -85,B 0,C 180,E1 26590.946,E2 26590.946} C_VEL
LIN {X 0,Y 552.333,Z 282,A -85,B 0,C 180,E1 26587.713,E2 26587.713} C_VEL
LIN {X 0,Y 552.32,Z 282.001,A -85,B 0,C 180,E1 26584.39,E2 26584.39} C_VEL
LIN {X 0,Y 552.314,Z 282.054,A -85,B 0,C 180,E1 26582.454,E2 26582.454} C_VEL
LIN {X 0,Y 556.713,Z 295.777,A -85,B 0,C 180,E1 26581.088,E2 26581.088} C_VEL
LIN {X 0,Y 555.919,Z 336.053,A -85,B 0,C 180,E1 26578.115,E2 26578.115} C_VEL
LIN {X 0,Y 555.27,Z 382.492,A -85,B 0,C 180,E1 26574.858,E2 26574.858} C_VEL
LIN {X 0,Y 555.308,Z 387.16,A -85,B 0,C 180,E1 26574.563,E2 26574.563} C_VEL
LIN {X 0,Y 556.408,Z 395.903,A -85,B 0,C 180,E1 26574.397,E2 26574.397} C_VEL
LIN {X 0,Y 555.434,Z 596.447,A -85,B 0,C 180,E1 26571.653,E2 26571.653} C_VEL
LIN {X 0,Y 555.166,Z 615.421,A -85,B 0,C 180,E1 26571.197,E2 26571.197} C_VEL
LIN {X 0,Y 554.834,Z 633.378,A -85,B 0,C 180,E1 26570.574,E2 26570.574} C_VEL
LIN {X 0,Y 554.429,Z 651.025,A -85,B 0,C 180,E1 26569.764,E2 26569.764} C_VEL
LIN {X 0,Y 554.002,Z 667.693,A -85,B 0,C 180,E1 26568.798,E2 26568.798} C_VEL
LIN {X 0,Y 553.575,Z 683.614,A -85,B 0,C 180,E1 26567.665,E2 26567.665} C_VEL
LIN {X 0,Y 553.164,Z 698.547,A -85,B 0,C 180,E1 26566.379,E2 26566.379} C_VEL
LIN {X 0,Y 552.809,Z 712.012,A -85,B 0,C 180,E1 26564.99,E2 26564.99} C_VEL
LIN {X 0,Y 552.499,Z 724.908,A -85,B 0,C 180,E1 26563.394,E2 26563.394} C_VEL
LIN {X 0,Y 552.266,Z 736.225,A -85,B 0,C 180,E1 26561.7,E2 26561.7} C_VEL
LIN {X 0,Y 552.097,Z 746.173,A -85,B 0,C 180,E1 26559.87,E2 26559.87} C_VEL
LIN {X 0,Y 551.991,Z 754.174,A -85,B 0,C 180,E1 26558.018,E2 26558.018} C_VEL
LIN {X 0,Y 551.939,Z 760.411,A -85,B 0,C 180,E1 26556.136,E2 26556.136} C_VEL
LIN {X 0,Y 551.914,Z 764.876,A -85,B 0,C 180,E1 26554.26,E2 26554.26} C_VEL
LIN {X 0,Y 551.912,Z 767.792,A -85,B 0,C 180,E1 26552.285,E2 26552.285} C_VEL
LIN {X 0,Y 551.908,Z 768.939,A -85,B 0,C 180,E1 26550.312,E2 26550.312} C_VEL
LIN {X 0,Y 551.913,Z 768.416,A -85,B 0,C 180,E1 26548.444,E2 26548.444} C_VEL
LIN {X 0,Y 551.91,Z 766.163,A -85,B 0,C 180,E1 26546.469,E2 26546.469} C_VEL
LIN {X 0,Y 551.93,Z 762.353,A -85,B 0,C 180,E1 26544.595,E2 26544.595} C_VEL
LIN {X 0,Y 551.97,Z 756.823,A -85,B 0,C 180,E1 26542.716,E2 26542.716} C_VEL
LIN {X 0,Y 552.055,Z 749.432,A -85,B 0,C 180,E1 26540.83,E2 26540.83} C_VEL
LIN {X 0,Y 552.183,Z 740.523,A -85,B 0,C 180,E1 26539.041,E2 26539.041} C_VEL
LIN {X 0,Y 552.39,Z 729.989,A -85,B 0,C 180,E1 26537.324,E2 26537.324} C_VEL
LIN {X 0,Y 552.654,Z 718.359,A -85,B 0,C 180,E1 26535.757,E2 26535.757} C_VEL
LIN {X 0,Y 553.007,Z 704.583,A -85,B 0,C 180,E1 26534.211,E2 26534.211} C_VEL
LIN {X 0,Y 553.415,Z 689.614,A -85,B 0,C 180,E1 26532.82,E2 26532.82} C_VEL
LIN {X 0,Y 553.854,Z 673.448,A -85,B 0,C 180,E1 26531.584,E2 26531.584} C_VEL
LIN {X 0,Y 554.275,Z 657.067,A -85,B 0,C 180,E1 26530.561,E2 26530.561} C_VEL
LIN {X 0,Y 554.689,Z 639.828,A -85,B 0,C 180,E1 26529.697,E2 26529.697} C_VEL
LIN {X 0,Y 555.06,Z 621.561,A -85,B 0,C 180,E1 26528.995,E2 26528.995} C_VEL
LIN {X 0,Y 555.35,Z 602.916,A -85,B 0,C 180,E1 26528.482,E2 26528.482} C_VEL
LIN {X 0,Y 555.532,Z 582.557,A -85,B 0,C 180,E1 26528.132,E2 26528.132} C_VEL
LIN {X 0,Y 556.253,Z 393.137,A -85,B 0,C 180,E1 26525.557,E2 26525.557} C_VEL
LIN {X 0,Y 555.245,Z 386.597,A -85,B 0,C 180,E1 26525.42,E2 26525.42} C_VEL
LIN {X 0,Y 556.118,Z 338.386,A -85,B 0,C 180,E1 26521.98,E2 26521.98} C_VEL
LIN {X 0,Y 556.859,Z 297.408,A -85,B 0,C 180,E1 26518.982,E2 26518.982} C_VEL
LIN {X 0,Y 556.603,Z 294.732,A -85,B 0,C 180,E1 26518.768,E2 26518.768} C_VEL
LIN {X 0,Y 552.307,Z 282.003,A -85,B 0,C 180,E1 26517.538,E2 26517.538} C_VEL
LIN {X 0,Y 552.269,Z 282.003,A -85,B 0,C 180,E1 26514.469,E2 26514.469} C_VEL
LIN {X 0,Y 552.268,Z 282.001,A -85,B 0,C 180,E1 26511.082,E2 26511.082} C_VEL
LIN {X 0,Y 552.317,Z 282.001,A -85,B 0,C 180,E1 26507.922,E2 26507.922} C_VEL
LIN {X 0,Y 552.258,Z 282.001,A -85,B 0,C 180,E1 26504.772,E2 26504.772} C_VEL
LIN {X 0,Y 552.324,Z 282,A -85,B 0,C 180,E1 26501.615,E2 26501.615} C_VEL
LIN {X 0,Y 552.262,Z 282,A -85,B 0,C 180,E1 26498.522,E2 26498.522} C_VEL
LIN {X 0,Y 552.276,Z 281.999,A -85,B 0,C 180,E1 26495.151,E2 26495.151} C_VEL
LIN {X 0,Y 552.298,Z 282,A -85,B 0,C 180,E1 26492.036,E2 26492.036} C_VEL
LIN {X 0,Y 552.263,Z 281.999,A -85,B 0,C 180,E1 26488.79,E2 26488.79} C_VEL
LIN {X 0,Y 552.333,Z 282,A -85,B 0,C 180,E1 26485.637,E2 26485.637} C_VEL
LIN {X 0,Y 552.266,Z 281.999,A -85,B 0,C 180,E1 26482.459,E2 26482.459} C_VEL
LIN {X 0,Y 552.28,Z 281.999,A -85,B 0,C 180,E1 26479.088,E2 26479.088} C_VEL
LIN {X 0,Y 552.302,Z 282,A -85,B 0,C 180,E1 26475.973,E2 26475.973} C_VEL
LIN {X 0,Y 552.266,Z 281.999,A -85,B 0,C 180,E1 26472.762,E2 26472.762} C_VEL
LIN {X 0,Y 552.335,Z 281.999,A -85,B 0,C 180,E1 26469.588,E2 26469.588} C_VEL
LIN {X 0,Y 552.269,Z 281.999,A -85,B 0,C 180,E1 26466.446,E2 26466.446} C_VEL
LIN {X 0,Y 552.292,Z 281.998,A -85,B 0,C 180,E1 26463.115,E2 26463.115} C_VEL
LIN {X 0,Y 552.296,Z 281.999,A -85,B 0,C 180,E1 26460.001,E2 26460.001} C_VEL
LIN {X 0,Y 552.272,Z 281.998,A -85,B 0,C 180,E1 26456.68,E2 26456.68} C_VEL
LIN {X 0,Y 552.337,Z 281.997,A -85,B 0,C 180,E1 26453.453,E2 26453.453} C_VEL
LIN {X 0,Y 552.276,Z 281.999,A -85,B 0,C 180,E1 26450.309,E2 26450.309} C_VEL
LIN {X 0,Y 552.285,Z 281.997,A -85,B 0,C 180,E1 26446.9,E2 26446.9} C_VEL
LIN {X 0,Y 552.313,Z 281.999,A -85,B 0,C 180,E1 26443.814,E2 26443.814} C_VEL
LIN {X 0,Y 552.275,Z 281.998,A -85,B 0,C 180,E1 26440.544,E2 26440.544} C_VEL
LIN {X 0,Y 552.336,Z 281.996,A -85,B 0,C 180,E1 26437.322,E2 26437.322} C_VEL
LIN {X 0,Y 552.286,Z 281.998,A -85,B 0,C 180,E1 26434.125,E2 26434.125} C_VEL
LIN {X 0,Y 552.286,Z 281.997,A -85,B 0,C 180,E1 26432.792,E2 26432.792} C_VEL
LIN {X 0,Y 551.295,Z 282.124,A -85,B 0,C 180,E1 26431.993,E2 26431.993} C_VEL
LIN {X 0,Y 544.86,Z 282.931,A -85,B 0,C 180,E1 26429.691,E2 26429.691} C_VEL
LIN {X 0,Y 544.383,Z 282.985,A -85,B 0,C 180,E1 26429.164,E2 26429.164} C_VEL
LIN {X 0,Y 544.361,Z 282.988,A -85,B 0,C 180,E1 26425.931,E2 26425.931} C_VEL
LIN {X 0,Y 544.342,Z 282.986,A -85,B 0,C 180,E1 26422.559,E2 26422.559} C_VEL
LIN {X 0,Y 544.407,Z 282.984,A -85,B 0,C 180,E1 26419.311,E2 26419.311} C_VEL
LIN {X 0,Y 544.351,Z 282.987,A -85,B 0,C 180,E1 26416.031,E2 26416.031} C_VEL
